Yaskawa INFORM job: A_ROOF_UPPER_0614_2_PAINT_36.JBI

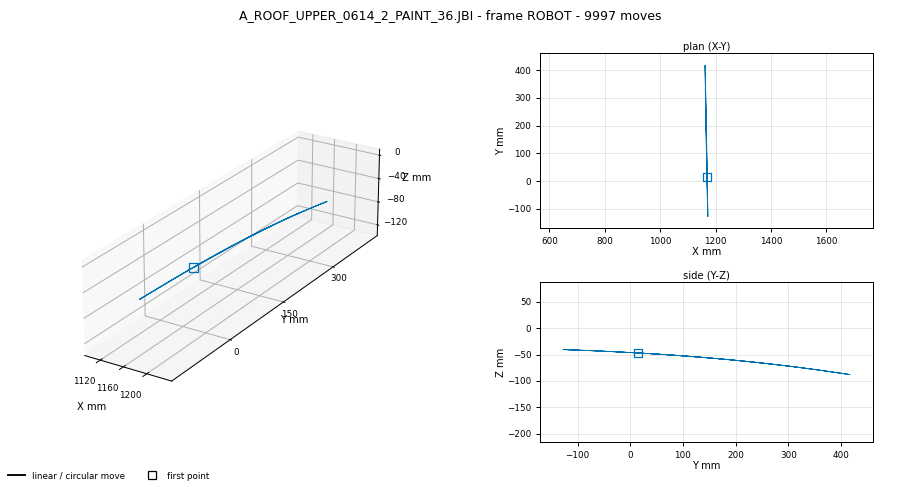
[picture p0: tool path of A_ROOF_UPPER_0614_2_PAINT_36.JBI in frame ROBOT, 9997 of 9997 moves have a stored position in this frame; points joined in program order, loops and branches not executed]
/JOB
//NAME A_ROOF_UPPER_0614_2_PAINT36
//POS
///NPOS 9997,0,0,0,0,0
///TOOL 1
///USER 0
///POSTYPE ROBOT
///RECTAN
///RCONF 1,0,0,0,0,0,0,0,0,0,0,0,0,0,0,0,0,0,0,0,0,0,0,0
C00000=1170.431,14.417,-46.796,-179.925,5.967,149.046
C00001=1170.426,14.666,-46.810,-179.923,5.968,149.045
C00002=1170.421,14.916,-46.824,-179.920,5.969,149.044
C00003=1170.416,15.166,-46.839,-179.918,5.970,149.044
C00004=1170.411,15.415,-46.853,-179.916,5.970,149.043
C00005=1170.405,15.664,-46.867,-179.913,5.970,149.043
C00006=1170.400,15.914,-46.881,-179.911,5.971,149.042
C00007=1170.396,16.164,-46.895,-179.908,5.973,149.042
C00008=1170.391,16.413,-46.910,-179.905,5.973,149.041
C00009=1170.386,16.663,-46.924,-179.903,5.974,149.040
C00010=1170.380,16.912,-46.938,-179.900,5.974,149.040
C00011=1170.375,17.161,-46.953,-179.898,5.975,149.039
C00012=1170.370,17.411,-46.967,-179.895,5.976,149.039
C00013=1170.366,17.661,-46.981,-179.893,5.977,149.038
C00014=1170.361,17.910,-46.996,-179.890,5.977,149.037
C00015=1170.356,18.160,-47.010,-179.887,5.978,149.037
C00016=1170.350,18.409,-47.024,-179.885,5.979,149.036
C00017=1170.345,18.659,-47.038,-179.882,5.980,149.036
C00018=1170.340,18.909,-47.052,-179.880,5.980,149.035
C00019=1170.334,19.159,-47.067,-179.878,5.981,149.034
C00020=1170.330,19.408,-47.082,-179.875,5.981,149.034
C00021=1170.325,19.657,-47.096,-179.873,5.982,149.033
C00022=1170.319,19.906,-47.110,-179.870,5.984,149.033
C00023=1170.314,20.156,-47.125,-179.867,5.984,149.032
C00024=1170.309,20.406,-47.139,-179.865,5.985,149.031
C00025=1170.304,20.656,-47.153,-179.862,5.985,149.031
C00026=1170.300,20.905,-47.168,-179.860,5.986,149.030
C00027=1170.295,21.154,-47.182,-179.857,5.987,149.030
C00028=1170.290,21.404,-47.197,-179.855,5.988,149.029
C00029=1170.284,21.653,-47.211,-179.852,5.989,149.029
C00030=1170.279,21.903,-47.226,-179.849,5.989,149.028
C00031=1170.274,22.152,-47.241,-179.847,5.990,149.027
C00032=1170.269,22.402,-47.255,-179.844,5.991,149.027
C00033=1170.264,22.652,-47.269,-179.842,5.991,149.026
C00034=1170.259,22.901,-47.283,-179.840,5.992,149.026
C00035=1170.254,23.151,-47.299,-179.836,5.993,149.025
C00036=1170.249,23.400,-47.313,-179.834,5.994,149.024
C00037=1170.244,23.650,-47.328,-179.832,5.995,149.024
C00038=1170.239,23.898,-47.342,-179.829,5.995,149.023
C00039=1170.234,24.148,-47.356,-179.827,5.996,149.023
C00040=1170.229,24.398,-47.371,-179.825,5.997,149.022
C00041=1170.223,24.647,-47.386,-179.821,5.998,149.022
C00042=1170.218,24.897,-47.401,-179.819,5.998,149.021
C00043=1170.213,25.147,-47.415,-179.817,5.999,149.020
C00044=1170.209,25.396,-47.430,-179.814,6.000,149.020
C00045=1170.203,25.646,-47.445,-179.812,6.001,149.019
C00046=1170.198,25.896,-47.459,-179.808,6.002,149.019
C00047=1170.193,26.145,-47.474,-179.806,6.002,149.018
C00048=1170.188,26.394,-47.488,-179.804,6.003,149.017
C00049=1170.183,26.644,-47.503,-179.801,6.004,149.017
C00050=1170.178,26.893,-47.518,-179.799,6.005,149.016
C00051=1170.173,27.143,-47.532,-179.796,6.006,149.016
C00052=1170.169,27.392,-47.547,-179.793,6.006,149.015
C00053=1170.163,27.642,-47.562,-179.791,6.007,149.015
C00054=1170.158,27.911,-47.578,-179.788,6.008,149.014
C00055=1170.153,28.180,-47.594,-179.785,6.009,149.013
C00056=1170.147,28.449,-47.610,-179.783,6.010,149.013
C00057=1170.141,28.717,-47.625,-179.780,6.010,149.012
C00058=1170.136,28.966,-47.640,-179.777,6.012,149.011
C00059=1170.131,29.216,-47.655,-179.775,6.012,149.011
C00060=1170.126,29.465,-47.670,-179.772,6.013,149.010
C00061=1170.121,29.715,-47.684,-179.769,6.013,149.010
C00062=1170.116,29.964,-47.700,-179.767,6.014,149.009
C00063=1170.111,30.215,-47.715,-179.764,6.016,149.008
C00064=1170.107,30.464,-47.730,-179.762,6.016,149.008
C00065=1170.101,30.714,-47.745,-179.759,6.017,149.007
C00066=1170.096,30.963,-47.760,-179.757,6.018,149.007
C00067=1170.091,31.213,-47.774,-179.754,6.018,149.006
C00068=1170.086,31.462,-47.789,-179.751,6.020,149.005
C00069=1170.081,31.712,-47.804,-179.749,6.020,149.005
C00070=1170.076,31.961,-47.819,-179.746,6.021,149.004
C00071=1170.071,32.210,-47.834,-179.744,6.022,149.004
C00072=1170.066,32.460,-47.849,-179.741,6.023,149.003
C00073=1170.061,32.709,-47.864,-179.739,6.024,149.003
C00074=1170.056,32.959,-47.878,-179.736,6.024,149.002
C00075=1170.050,33.209,-47.894,-179.734,6.025,149.001
C00076=1170.046,33.458,-47.909,-179.731,6.026,149.001
C00077=1170.040,33.708,-47.924,-179.728,6.027,149.000
C00078=1170.035,33.957,-47.939,-179.726,6.028,149.000
C00079=1170.031,34.206,-47.954,-179.723,6.028,148.999
C00080=1170.025,34.456,-47.969,-179.721,6.029,148.999
C00081=1170.021,34.706,-47.984,-179.718,6.030,148.998
C00082=1170.016,34.955,-48.000,-179.715,6.031,148.997
C00083=1170.011,35.205,-48.014,-179.713,6.032,148.997
C00084=1170.005,35.454,-48.030,-179.710,6.032,148.996
C00085=1170.001,35.703,-48.045,-179.708,6.034,148.996
C00086=1169.995,35.953,-48.060,-179.705,6.034,148.995
C00087=1169.990,36.202,-48.074,-179.703,6.035,148.995
C00088=1169.985,36.452,-48.090,-179.700,6.036,148.994
C00089=1169.980,36.701,-48.105,-179.698,6.037,148.994
C00090=1169.975,36.951,-48.121,-179.695,6.038,148.993
C00091=1169.970,37.201,-48.135,-179.692,6.038,148.992
C00092=1169.965,37.450,-48.151,-179.690,6.039,148.992
C00093=1169.960,37.699,-48.166,-179.687,6.041,148.991
C00094=1169.955,37.949,-48.181,-179.685,6.041,148.991
C00095=1169.950,38.198,-48.196,-179.682,6.042,148.990
C00096=1169.945,38.448,-48.211,-179.680,6.043,148.990
C00097=1169.940,38.698,-48.227,-179.677,6.044,148.989
C00098=1169.935,38.947,-48.242,-179.674,6.045,148.988
C00099=1169.930,39.196,-48.258,-179.672,6.045,148.988
C00100=1169.925,39.445,-48.273,-179.669,6.046,148.987
C00101=1169.920,39.695,-48.288,-179.666,6.048,148.987
C00102=1169.915,39.944,-48.303,-179.664,6.048,148.986
C00103=1169.910,40.195,-48.319,-179.662,6.049,148.985
C00104=1169.905,40.444,-48.334,-179.659,6.049,148.985
C00105=1169.900,40.693,-48.349,-179.656,6.051,148.984
C00106=1169.895,40.942,-48.365,-179.654,6.052,148.984
C00107=1169.889,41.192,-48.380,-179.652,6.052,148.983
C00108=1169.885,41.441,-48.395,-179.648,6.054,148.983
C00109=1169.880,41.691,-48.411,-179.646,6.054,148.982
C00110=1169.875,41.940,-48.426,-179.643,6.055,148.981
C00111=1169.870,42.190,-48.442,-179.641,6.056,148.981
C00112=1169.864,42.439,-48.457,-179.638,6.057,148.980
C00113=1169.860,42.689,-48.473,-179.635,6.058,148.980
C00114=1169.855,42.938,-48.488,-179.633,6.059,148.979
C00115=1169.849,43.188,-48.503,-179.630,6.060,148.979
C00116=1169.845,43.437,-48.518,-179.628,6.061,148.978
C00117=1169.840,43.686,-48.535,-179.625,6.061,148.977
C00118=1169.835,43.936,-48.551,-179.623,6.062,148.977
C00119=1169.830,44.185,-48.565,-179.620,6.063,148.976
C00120=1169.825,44.435,-48.581,-179.617,6.064,148.976
C00121=1169.819,44.684,-48.597,-179.615,6.065,148.975
C00122=1169.815,44.934,-48.613,-179.612,6.066,148.975
C00123=1169.810,45.183,-48.628,-179.610,6.067,148.974
C00124=1169.804,45.433,-48.643,-179.607,6.067,148.973
C00125=1169.800,45.683,-48.659,-179.605,6.068,148.973
C00126=1169.794,45.932,-48.675,-179.602,6.070,148.972
C00127=1169.790,46.181,-48.690,-179.600,6.071,148.972
C00128=1169.784,46.431,-48.705,-179.597,6.071,148.971
C00129=1169.779,46.681,-48.721,-179.594,6.073,148.971
C00130=1169.774,46.930,-48.737,-179.591,6.073,148.970
C00131=1169.770,47.179,-48.753,-179.589,6.074,148.970
C00132=1169.765,47.429,-48.769,-179.586,6.075,148.969
C00133=1169.760,47.678,-48.784,-179.583,6.076,148.968
C00134=1169.754,47.928,-48.800,-179.581,6.077,148.968
C00135=1169.750,48.177,-48.815,-179.578,6.078,148.967
C00136=1169.745,48.427,-48.831,-179.576,6.079,148.967
C00137=1169.740,48.676,-48.847,-179.573,6.079,148.966
C00138=1169.735,48.926,-48.863,-179.571,6.081,148.966
C00139=1169.730,49.175,-48.878,-179.568,6.082,148.965
C00140=1169.725,49.424,-48.893,-179.566,6.082,148.965
C00141=1169.720,49.674,-48.909,-179.563,6.084,148.964
C00142=1169.715,49.923,-48.926,-179.560,6.085,148.963
C00143=1169.710,50.172,-48.941,-179.558,6.085,148.963
C00144=1169.705,50.423,-48.957,-179.555,6.087,148.962
C00145=1169.699,50.672,-48.973,-179.552,6.087,148.962
C00146=1169.694,50.921,-48.989,-179.550,6.088,148.961
C00147=1169.690,51.171,-49.005,-179.547,6.089,148.961
C00148=1169.685,51.420,-49.020,-179.545,6.090,148.960
C00149=1169.680,51.669,-49.037,-179.542,6.091,148.959
C00150=1169.675,51.919,-49.052,-179.539,6.092,148.959
C00151=1169.670,52.168,-49.068,-179.537,6.093,148.958
C00152=1169.665,52.418,-49.085,-179.534,6.093,148.958
C00153=1169.660,52.667,-49.100,-179.531,6.095,148.957
C00154=1169.654,52.916,-49.116,-179.529,6.096,148.957
C00155=1169.650,53.166,-49.132,-179.527,6.097,148.956
C00156=1169.645,53.415,-49.148,-179.523,6.098,148.955
C00157=1169.640,53.665,-49.164,-179.521,6.099,148.955
C00158=1169.634,53.934,-49.181,-179.518,6.100,148.954
C00159=1169.629,54.202,-49.199,-179.515,6.101,148.954
C00160=1169.623,54.470,-49.216,-179.513,6.102,148.953
C00161=1169.618,54.739,-49.233,-179.510,6.103,148.953
C00162=1169.613,54.989,-49.249,-179.507,6.104,148.952
C00163=1169.609,55.238,-49.265,-179.505,6.105,148.951
C00164=1169.603,55.488,-49.281,-179.502,6.106,148.951
C00165=1169.598,55.737,-49.297,-179.499,6.107,148.950
C00166=1169.593,55.987,-49.313,-179.497,6.108,148.950
C00167=1169.588,56.235,-49.330,-179.494,6.108,148.949
C00168=1169.583,56.486,-49.346,-179.492,6.110,148.949
C00169=1169.578,56.734,-49.362,-179.489,6.111,148.948
C00170=1169.574,56.984,-49.378,-179.487,6.112,148.948
C00171=1169.568,57.233,-49.394,-179.484,6.113,148.947
C00172=1169.564,57.483,-49.410,-179.482,6.114,148.947
C00173=1169.559,57.732,-49.426,-179.478,6.115,148.946
C00174=1169.554,57.982,-49.442,-179.476,6.116,148.946
C00175=1169.549,58.231,-49.459,-179.474,6.116,148.945
C00176=1169.544,58.481,-49.475,-179.471,6.118,148.944
C00177=1169.539,58.730,-49.491,-179.468,6.119,148.944
C00178=1169.534,58.980,-49.507,-179.465,6.120,148.943
C00179=1169.529,59.229,-49.523,-179.463,6.121,148.943
C00180=1169.525,59.478,-49.540,-179.461,6.122,148.942
C00181=1169.519,59.728,-49.555,-179.457,6.123,148.942
C00182=1169.515,59.977,-49.572,-179.455,6.124,148.941
C00183=1169.509,60.227,-49.588,-179.453,6.124,148.940
C00184=1169.504,60.476,-49.605,-179.450,6.126,148.940
C00185=1169.499,60.725,-49.621,-179.447,6.127,148.939
C00186=1169.494,60.975,-49.637,-179.445,6.128,148.939
C00187=1169.489,61.224,-49.653,-179.442,6.129,148.938
C00188=1169.485,61.473,-49.670,-179.440,6.130,148.938
C00189=1169.479,61.723,-49.686,-179.437,6.131,148.937
C00190=1169.474,61.973,-49.703,-179.434,6.132,148.937
C00191=1169.469,62.221,-49.719,-179.431,6.133,148.936
C00192=1169.464,62.472,-49.735,-179.429,6.134,148.936
C00193=1169.460,62.721,-49.752,-179.426,6.135,148.935
C00194=1169.455,62.970,-49.768,-179.424,6.136,148.935
C00195=1169.450,63.219,-49.785,-179.421,6.137,148.934
C00196=1169.444,63.469,-49.801,-179.418,6.138,148.933
C00197=1169.440,63.719,-49.818,-179.416,6.139,148.933
C00198=1169.434,63.967,-49.834,-179.413,6.141,148.932
C00199=1169.430,64.217,-49.851,-179.410,6.141,148.932
C00200=1169.425,64.467,-49.867,-179.408,6.142,148.931
C00201=1169.419,64.716,-49.884,-179.405,6.143,148.931
C00202=1169.415,64.965,-49.900,-179.403,6.144,148.930
C00203=1169.410,65.215,-49.917,-179.400,6.145,148.929
C00204=1169.405,65.464,-49.933,-179.397,6.146,148.929
C00205=1169.400,65.714,-49.950,-179.394,6.148,148.928
C00206=1169.395,65.963,-49.966,-179.392,6.149,148.928
C00207=1169.390,66.212,-49.983,-179.390,6.149,148.927
C00208=1169.386,66.462,-49.999,-179.387,6.151,148.927
C00209=1169.380,66.711,-50.016,-179.385,6.152,148.926
C00210=1169.375,66.960,-50.033,-179.381,6.153,148.926
C00211=1169.371,67.210,-50.050,-179.379,6.154,148.925
C00212=1169.365,67.460,-50.066,-179.376,6.155,148.925
C00213=1169.360,67.709,-50.082,-179.374,6.156,148.924
C00214=1169.356,67.959,-50.099,-179.371,6.157,148.924
C00215=1169.351,68.207,-50.115,-179.368,6.158,148.923
C00216=1169.346,68.457,-50.133,-179.366,6.159,148.922
C00217=1169.341,68.707,-50.149,-179.363,6.160,148.922
C00218=1169.336,68.955,-50.166,-179.360,6.161,148.921
C00219=1169.331,69.205,-50.183,-179.358,6.163,148.921
C00220=1169.326,69.455,-50.200,-179.355,6.163,148.920
C00221=1169.321,69.704,-50.217,-179.352,6.165,148.920
C00222=1169.316,69.953,-50.233,-179.350,6.166,148.919
C00223=1169.312,70.203,-50.250,-179.347,6.167,148.919
C00224=1169.306,70.452,-50.267,-179.345,6.168,148.918
C00225=1169.301,70.701,-50.283,-179.342,6.168,148.918
C00226=1169.297,70.951,-50.300,-179.339,6.170,148.917
C00227=1169.291,71.200,-50.317,-179.337,6.171,148.917
C00228=1169.286,71.449,-50.334,-179.334,6.172,148.916
C00229=1169.281,71.699,-50.351,-179.331,6.173,148.915
C00230=1169.277,71.949,-50.368,-179.329,6.175,148.915
C00231=1169.271,72.198,-50.384,-179.326,6.175,148.914
C00232=1169.266,72.447,-50.401,-179.323,6.177,148.914
C00233=1169.262,72.697,-50.418,-179.321,6.178,148.914
C00234=1169.257,72.946,-50.436,-179.318,6.179,148.913
C00235=1169.252,73.195,-50.452,-179.316,6.180,148.912
C00236=1169.247,73.445,-50.469,-179.313,6.181,148.912
C00237=1169.242,73.694,-50.486,-179.310,6.182,148.911
C00238=1169.237,73.944,-50.503,-179.307,6.183,148.911
C00239=1169.232,74.193,-50.520,-179.305,6.184,148.910
C00240=1169.227,74.442,-50.537,-179.302,6.186,148.910
C00241=1169.223,74.691,-50.554,-179.300,6.186,148.909
C00242=1169.217,74.941,-50.572,-179.297,6.188,148.909
C00243=1169.212,75.190,-50.588,-179.294,6.189,148.908
C00244=1169.207,75.440,-50.605,-179.292,6.190,148.908
C00245=1169.203,75.689,-50.622,-179.289,6.191,148.907
C00246=1169.198,75.938,-50.640,-179.286,6.193,148.907
C00247=1169.193,76.188,-50.656,-179.284,6.193,148.906
C00248=1169.187,76.437,-50.673,-179.281,6.195,148.906
C00249=1169.183,76.686,-50.690,-179.279,6.196,148.905
C00250=1169.178,76.936,-50.708,-179.276,6.197,148.904
C00251=1169.174,77.185,-50.725,-179.273,6.198,148.904
C00252=1169.168,77.435,-50.742,-179.270,6.199,148.903
C00253=1169.163,77.685,-50.759,-179.268,6.200,148.903
C00254=1169.158,77.933,-50.776,-179.265,6.201,148.902
C00255=1169.153,78.183,-50.793,-179.263,6.202,148.902
C00256=1169.149,78.432,-50.810,-179.260,6.204,148.901
C00257=1169.144,78.681,-50.828,-179.257,6.205,148.901
C00258=1169.139,78.931,-50.845,-179.255,6.206,148.900
C00259=1169.134,79.181,-50.862,-179.252,6.207,148.900
C00260=1169.129,79.429,-50.880,-179.249,6.208,148.899
C00261=1169.124,79.678,-50.896,-179.247,6.209,148.899
C00262=1169.119,79.947,-50.915,-179.244,6.211,148.898
C00263=1169.114,80.216,-50.934,-179.241,6.212,148.898
C00264=1169.108,80.484,-50.953,-179.239,6.213,148.897
C00265=1169.103,80.752,-50.971,-179.235,6.214,148.896
C00266=1169.098,81.002,-50.989,-179.233,6.216,148.896
C00267=1169.093,81.251,-51.006,-179.230,6.216,148.895
C00268=1169.088,81.501,-51.023,-179.227,6.218,148.895
C00269=1169.083,81.750,-51.041,-179.225,6.219,148.894
C00270=1169.078,82.000,-51.058,-179.222,6.220,148.894
C00271=1169.073,82.248,-51.075,-179.220,6.221,148.893
C00272=1169.068,82.498,-51.092,-179.217,6.223,148.893
C00273=1169.063,82.747,-51.110,-179.214,6.223,148.892
C00274=1169.058,82.997,-51.128,-179.211,6.225,148.892
C00275=1169.054,83.246,-51.145,-179.209,6.226,148.891
C00276=1169.049,83.495,-51.162,-179.206,6.227,148.891
C00277=1169.044,83.745,-51.180,-179.203,6.229,148.890
C00278=1169.039,83.994,-51.197,-179.201,6.230,148.890
C00279=1169.034,84.243,-51.215,-179.198,6.231,148.889
C00280=1169.029,84.493,-51.232,-179.196,6.232,148.889
C00281=1169.024,84.742,-51.250,-179.193,6.234,148.888
C00282=1169.019,84.991,-51.268,-179.190,6.234,148.888
C00283=1169.015,85.241,-51.285,-179.188,6.236,148.887
C00284=1169.010,85.490,-51.303,-179.185,6.237,148.887
C00285=1169.005,85.740,-51.320,-179.182,6.238,148.886
C00286=1169.000,85.989,-51.338,-179.179,6.240,148.886
C00287=1168.995,86.238,-51.356,-179.177,6.240,148.885
C00288=1168.990,86.488,-51.373,-179.174,6.242,148.885
C00289=1168.985,86.737,-51.391,-179.172,6.243,148.884
C00290=1168.981,86.986,-51.409,-179.169,6.244,148.884
C00291=1168.975,87.236,-51.426,-179.167,6.245,148.883
C00292=1168.970,87.485,-51.444,-179.163,6.246,148.883
C00293=1168.966,87.734,-51.462,-179.161,6.248,148.882
C00294=1168.961,87.984,-51.478,-179.159,6.249,148.882
C00295=1168.956,88.233,-51.496,-179.155,6.250,148.881
C00296=1168.951,88.482,-51.514,-179.153,6.251,148.881
C00297=1168.946,88.732,-51.532,-179.151,6.253,148.880
C00298=1168.941,88.981,-51.550,-179.148,6.253,148.880
C00299=1168.936,89.230,-51.568,-179.145,6.255,148.879
C00300=1168.931,89.479,-51.586,-179.142,6.256,148.878
C00301=1168.926,89.729,-51.603,-179.140,6.257,148.878
C00302=1168.922,89.978,-51.620,-179.137,6.259,148.878
C00303=1168.917,90.227,-51.638,-179.134,6.260,148.877
C00304=1168.912,90.476,-51.656,-179.132,6.261,148.877
C00305=1168.907,90.725,-51.674,-179.129,6.263,148.876
C00306=1168.902,90.975,-51.691,-179.126,6.264,148.876
C00307=1168.897,91.224,-51.709,-179.124,6.265,148.875
C00308=1168.892,91.474,-51.727,-179.121,6.266,148.874
C00309=1168.887,91.723,-51.745,-179.118,6.267,148.874
C00310=1168.882,91.972,-51.763,-179.116,6.269,148.874
C00311=1168.877,92.221,-51.781,-179.113,6.270,148.873
C00312=1168.872,92.471,-51.799,-179.110,6.271,148.873
C00313=1168.868,92.721,-51.817,-179.108,6.272,148.872
C00314=1168.863,92.970,-51.835,-179.105,6.274,148.871
C00315=1168.858,93.219,-51.853,-179.102,6.275,148.871
C00316=1168.853,93.468,-51.871,-179.100,6.276,148.871
C00317=1168.848,93.718,-51.889,-179.097,6.278,148.870
C00318=1168.843,93.967,-51.907,-179.095,6.278,148.870
C00319=1168.838,94.216,-51.925,-179.092,6.280,148.869
C00320=1168.833,94.465,-51.943,-179.089,6.282,148.869
C00321=1168.829,94.714,-51.961,-179.087,6.282,148.868
C00322=1168.824,94.964,-51.979,-179.084,6.284,148.868
C00323=1168.819,95.213,-51.997,-179.081,6.285,148.867
C00324=1168.814,95.462,-52.015,-179.079,6.286,148.867
C00325=1168.810,95.712,-52.033,-179.075,6.288,148.866
C00326=1168.805,95.961,-52.051,-179.073,6.289,148.866
C00327=1168.800,96.210,-52.069,-179.071,6.290,148.865
C00328=1168.794,96.459,-52.088,-179.067,6.292,148.865
C00329=1168.790,96.709,-52.106,-179.065,6.293,148.864
C00330=1168.785,96.959,-52.124,-179.062,6.294,148.864
C00331=1168.780,97.208,-52.142,-179.059,6.296,148.863
C00332=1168.775,97.457,-52.160,-179.057,6.297,148.863
C00333=1168.770,97.706,-52.178,-179.054,6.298,148.862
C00334=1168.766,97.956,-52.196,-179.051,6.300,148.862
C00335=1168.761,98.205,-52.214,-179.049,6.300,148.861
C00336=1168.755,98.455,-52.233,-179.046,6.302,148.861
C00337=1168.751,98.703,-52.251,-179.044,6.303,148.860
C00338=1168.746,98.952,-52.269,-179.041,6.304,148.860
C00339=1168.741,99.202,-52.288,-179.038,6.306,148.859
C00340=1168.736,99.451,-52.306,-179.036,6.307,148.859
C00341=1168.732,99.701,-52.324,-179.033,6.308,148.858
C00342=1168.726,99.950,-52.342,-179.030,6.310,148.858
C00343=1168.721,100.199,-52.361,-179.028,6.311,148.857
C00344=1168.717,100.448,-52.379,-179.025,6.312,148.857
C00345=1168.712,100.698,-52.397,-179.022,6.314,148.856
C00346=1168.707,100.947,-52.415,-179.020,6.315,148.856
C00347=1168.702,101.196,-52.434,-179.017,6.316,148.855
C00348=1168.697,101.446,-52.453,-179.014,6.318,148.855
C00349=1168.693,101.695,-52.471,-179.012,6.319,148.854
C00350=1168.688,101.944,-52.489,-179.009,6.320,148.854
C00351=1168.682,102.193,-52.508,-179.006,6.322,148.853
C00352=1168.678,102.443,-52.527,-179.004,6.323,148.853
C00353=1168.673,102.692,-52.545,-179.001,6.324,148.852
C00354=1168.668,102.941,-52.563,-178.998,6.326,148.852
C00355=1168.663,103.191,-52.582,-178.996,6.327,148.851
C00356=1168.659,103.440,-52.600,-178.993,6.328,148.851
C00357=1168.654,103.689,-52.618,-178.990,6.330,148.850
C00358=1168.649,103.937,-52.637,-178.988,6.331,148.850
C00359=1168.644,104.188,-52.656,-178.985,6.333,148.850
C00360=1168.639,104.437,-52.674,-178.982,6.334,148.849
C00361=1168.634,104.685,-52.692,-178.979,6.336,148.849
C00362=1168.629,104.936,-52.711,-178.977,6.337,148.848
C00363=1168.624,105.185,-52.729,-178.974,6.338,148.848
C00364=1168.620,105.433,-52.748,-178.971,6.340,148.847
C00365=1168.615,105.684,-52.767,-178.969,6.340,148.847
C00366=1168.610,105.951,-52.787,-178.966,6.342,148.846
C00367=1168.604,106.220,-52.807,-178.963,6.344,148.846
C00368=1168.599,106.488,-52.827,-178.960,6.345,148.845
C00369=1168.594,106.757,-52.848,-178.957,6.347,148.845
C00370=1168.589,107.006,-52.866,-178.954,6.348,148.844
C00371=1168.584,107.255,-52.885,-178.952,6.349,148.844
C00372=1168.580,107.505,-52.903,-178.949,6.351,148.843
C00373=1168.575,107.754,-52.921,-178.946,6.352,148.843
C00374=1168.570,108.003,-52.941,-178.944,6.353,148.842
C00375=1168.565,108.252,-52.960,-178.941,6.355,148.842
C00376=1168.560,108.501,-52.978,-178.938,6.356,148.841
C00377=1168.556,108.751,-52.997,-178.936,6.358,148.841
C00378=1168.550,109.000,-53.016,-178.933,6.359,148.840
C00379=1168.546,109.249,-53.034,-178.930,6.360,148.840
C00380=1168.540,109.499,-53.053,-178.928,6.362,148.839
C00381=1168.536,109.747,-53.072,-178.925,6.364,148.839
C00382=1168.532,109.997,-53.090,-178.922,6.364,148.838
C00383=1168.526,110.246,-53.110,-178.920,6.366,148.838
C00384=1168.522,110.495,-53.128,-178.917,6.368,148.838
C00385=1168.517,110.745,-53.147,-178.915,6.369,148.837
C00386=1168.512,110.993,-53.166,-178.911,6.370,148.837
C00387=1168.507,111.243,-53.186,-178.909,6.372,148.836
C00388=1168.502,111.492,-53.204,-178.906,6.373,148.836
C00389=1168.498,111.742,-53.223,-178.903,6.374,148.835
C00390=1168.493,111.990,-53.242,-178.901,6.376,148.835
C00391=1168.488,112.240,-53.261,-178.898,6.377,148.834
C00392=1168.483,112.489,-53.280,-178.895,6.379,148.834
C00393=1168.478,112.738,-53.299,-178.893,6.380,148.833
C00394=1168.473,112.988,-53.318,-178.890,6.381,148.833
C00395=1168.468,113.237,-53.337,-178.887,6.383,148.832
C00396=1168.464,113.486,-53.356,-178.885,6.385,148.832
C00397=1168.459,113.735,-53.374,-178.882,6.385,148.831
C00398=1168.454,113.985,-53.394,-178.879,6.387,148.831
C00399=1168.449,114.234,-53.413,-178.876,6.389,148.831
C00400=1168.445,114.483,-53.432,-178.874,6.391,148.830
C00401=1168.439,114.732,-53.452,-178.872,6.391,148.830
C00402=1168.435,114.982,-53.470,-178.868,6.393,148.829
C00403=1168.430,115.231,-53.489,-178.866,6.395,148.829
C00404=1168.425,115.480,-53.509,-178.863,6.396,148.828
C00405=1168.420,115.729,-53.528,-178.861,6.397,148.828
C00406=1168.415,115.978,-53.547,-178.858,6.399,148.827
C00407=1168.410,116.228,-53.566,-178.855,6.400,148.827
C00408=1168.406,116.477,-53.585,-178.852,6.402,148.826
C00409=1168.400,116.726,-53.604,-178.850,6.403,148.826
C00410=1168.396,116.976,-53.624,-178.847,6.404,148.825
C00411=1168.391,117.224,-53.642,-178.844,6.406,148.825
C00412=1168.386,117.474,-53.662,-178.842,6.408,148.825
C00413=1168.381,117.723,-53.681,-178.839,6.409,148.824
C00414=1168.377,117.972,-53.701,-178.836,6.410,148.824
C00415=1168.372,118.221,-53.720,-178.833,6.412,148.823
C00416=1168.367,118.470,-53.739,-178.831,6.413,148.823
C00417=1168.362,118.720,-53.759,-178.828,6.415,148.822
C00418=1168.358,118.968,-53.778,-178.825,6.417,148.822
C00419=1168.353,119.219,-53.797,-178.823,6.417,148.821
C00420=1168.347,119.467,-53.816,-178.820,6.419,148.821
C00421=1168.343,119.717,-53.835,-178.817,6.421,148.821
C00422=1168.338,119.966,-53.855,-178.815,6.423,148.820
C00423=1168.333,120.215,-53.874,-178.812,6.423,148.820
C00424=1168.329,120.464,-53.894,-178.809,6.425,148.819
C00425=1168.323,120.713,-53.914,-178.807,6.427,148.819
C00426=1168.319,120.962,-53.933,-178.804,6.428,148.818
C00427=1168.315,121.212,-53.952,-178.801,6.430,148.818
C00428=1168.309,121.461,-53.972,-178.798,6.432,148.818
C00429=1168.304,121.710,-53.991,-178.796,6.432,148.817
C00430=1168.300,121.960,-54.011,-178.793,6.434,148.817
C00431=1168.295,122.208,-54.030,-178.790,6.436,148.816
C00432=1168.290,122.458,-54.049,-178.788,6.437,148.816
C00433=1168.285,122.707,-54.069,-178.785,6.439,148.815
C00434=1168.280,122.956,-54.088,-178.782,6.440,148.815
C00435=1168.276,123.205,-54.109,-178.780,6.441,148.814
C00436=1168.271,123.454,-54.128,-178.777,6.443,148.814
C00437=1168.266,123.703,-54.147,-178.774,6.445,148.813
C00438=1168.262,123.953,-54.167,-178.772,6.447,148.813
C00439=1168.256,124.202,-54.186,-178.769,6.447,148.812
C00440=1168.252,124.451,-54.206,-178.766,6.449,148.812
C00441=1168.247,124.700,-54.226,-178.764,6.451,148.812
C00442=1168.242,124.949,-54.245,-178.761,6.452,148.811
C00443=1168.237,125.199,-54.265,-178.758,6.454,148.811
C00444=1168.232,125.448,-54.285,-178.755,6.456,148.810
C00445=1168.228,125.697,-54.305,-178.753,6.456,148.810
C00446=1168.223,125.946,-54.324,-178.750,6.458,148.809
C00447=1168.219,126.195,-54.343,-178.747,6.460,148.809
C00448=1168.214,126.445,-54.363,-178.745,6.462,148.809
C00449=1168.209,126.693,-54.383,-178.742,6.463,148.808
C00450=1168.204,126.943,-54.403,-178.739,6.465,148.808
C00451=1168.199,127.192,-54.422,-178.736,6.466,148.807
C00452=1168.195,127.441,-54.443,-178.734,6.467,148.807
C00453=1168.190,127.690,-54.462,-178.731,6.469,148.806
C00454=1168.185,127.940,-54.482,-178.729,6.471,148.806
C00455=1168.180,128.189,-54.502,-178.726,6.473,148.806
C00456=1168.176,128.438,-54.522,-178.723,6.474,148.805
C00457=1168.170,128.687,-54.541,-178.720,6.476,148.805
C00458=1168.166,128.936,-54.561,-178.718,6.477,148.804
C00459=1168.161,129.186,-54.581,-178.715,6.478,148.804
C00460=1168.157,129.435,-54.601,-178.712,6.480,148.803
C00461=1168.151,129.683,-54.621,-178.710,6.482,148.803
C00462=1168.147,129.933,-54.640,-178.707,6.483,148.802
C00463=1168.142,130.182,-54.661,-178.704,6.485,148.802
C00464=1168.137,130.432,-54.680,-178.701,6.487,148.802
C00465=1168.133,130.680,-54.701,-178.698,6.488,148.801
C00466=1168.127,130.930,-54.721,-178.696,6.489,148.801
C00467=1168.122,131.179,-54.741,-178.694,6.491,148.800
C00468=1168.118,131.428,-54.761,-178.691,6.493,148.800
C00469=1168.113,131.677,-54.781,-178.688,6.494,148.799
C00470=1168.108,131.946,-54.802,-178.685,6.496,148.799
C00471=1168.103,132.215,-54.824,-178.682,6.498,148.799
C00472=1168.098,132.483,-54.846,-178.680,6.499,148.798
C00473=1168.092,132.752,-54.867,-178.676,6.501,148.798
C00474=1168.088,133.001,-54.888,-178.674,6.502,148.797
C00475=1168.083,133.250,-54.907,-178.671,6.504,148.797
C00476=1168.078,133.498,-54.927,-178.668,6.506,148.796
C00477=1168.073,133.748,-54.947,-178.666,6.508,148.796
C00478=1168.069,133.997,-54.967,-178.663,6.509,148.796
C00479=1168.064,134.246,-54.988,-178.660,6.511,148.795
C00480=1168.059,134.496,-55.008,-178.657,6.512,148.795
C00481=1168.055,134.745,-55.028,-178.654,6.514,148.794
C00482=1168.050,134.993,-55.048,-178.652,6.516,148.794
C00483=1168.045,135.243,-55.068,-178.649,6.517,148.794
C00484=1168.040,135.492,-55.089,-178.647,6.519,148.793
C00485=1168.035,135.741,-55.109,-178.644,6.520,148.793
C00486=1168.031,135.990,-55.129,-178.641,6.522,148.792
C00487=1168.026,136.239,-55.149,-178.639,6.524,148.792
C00488=1168.021,136.489,-55.170,-178.635,6.525,148.791
C00489=1168.016,136.738,-55.190,-178.633,6.527,148.791
C00490=1168.012,136.987,-55.210,-178.630,6.529,148.791
C00491=1168.007,137.235,-55.230,-178.627,6.530,148.790
C00492=1168.002,137.485,-55.251,-178.625,6.532,148.790
C00493=1167.997,137.734,-55.271,-178.622,6.534,148.789
C00494=1167.992,137.983,-55.291,-178.620,6.535,148.789
C00495=1167.988,138.232,-55.312,-178.617,6.536,148.789
C00496=1167.983,138.481,-55.333,-178.614,6.538,148.788
C00497=1167.978,138.730,-55.353,-178.612,6.540,148.788
C00498=1167.974,138.980,-55.373,-178.609,6.541,148.787
C00499=1167.968,139.229,-55.394,-178.606,6.543,148.787
C00500=1167.964,139.478,-55.414,-178.603,6.545,148.786
C00501=1167.960,139.727,-55.434,-178.600,6.547,148.786
C00502=1167.954,139.976,-55.455,-178.598,6.548,148.786
C00503=1167.950,140.225,-55.476,-178.595,6.550,148.785
C00504=1167.945,140.474,-55.496,-178.592,6.552,148.785
C00505=1167.940,140.724,-55.516,-178.590,6.554,148.785
C00506=1167.936,140.973,-55.537,-178.587,6.555,148.784
C00507=1167.931,141.222,-55.557,-178.584,6.557,148.784
C00508=1167.926,141.471,-55.578,-178.581,6.559,148.783
C00509=1167.922,141.720,-55.598,-178.579,6.560,148.783
C00510=1167.916,141.969,-55.619,-178.576,6.561,148.782
C00511=1167.912,142.218,-55.640,-178.573,6.563,148.782
C00512=1167.907,142.467,-55.660,-178.571,6.565,148.782
C00513=1167.902,142.717,-55.681,-178.568,6.566,148.781
C00514=1167.898,142.966,-55.701,-178.565,6.568,148.781
C00515=1167.893,143.215,-55.722,-178.563,6.570,148.780
C00516=1167.888,143.464,-55.743,-178.560,6.571,148.780
C00517=1167.883,143.713,-55.764,-178.557,6.573,148.780
C00518=1167.879,143.962,-55.784,-178.555,6.575,148.779
C00519=1167.874,144.211,-55.805,-178.552,6.577,148.779
C00520=1167.869,144.460,-55.826,-178.549,6.578,148.778
C00521=1167.865,144.709,-55.846,-178.546,6.580,148.778
C00522=1167.859,144.958,-55.867,-178.544,6.582,148.778
C00523=1167.855,145.207,-55.888,-178.541,6.584,148.777
C00524=1167.850,145.456,-55.909,-178.538,6.585,148.777
C00525=1167.846,145.706,-55.930,-178.536,6.587,148.777
C00526=1167.841,145.955,-55.951,-178.533,6.589,148.776
C00527=1167.837,146.204,-55.971,-178.530,6.590,148.776
C00528=1167.831,146.453,-55.992,-178.527,6.592,148.775
C00529=1167.826,146.702,-56.013,-178.524,6.594,148.775
C00530=1167.822,146.951,-56.033,-178.522,6.595,148.774
C00531=1167.817,147.200,-56.055,-178.519,6.597,148.774
C00532=1167.813,147.449,-56.075,-178.516,6.599,148.774
C00533=1167.807,147.698,-56.096,-178.514,6.601,148.773
C00534=1167.803,147.947,-56.117,-178.511,6.602,148.773
C00535=1167.799,148.196,-56.139,-178.508,6.604,148.773
C00536=1167.794,148.446,-56.160,-178.506,6.606,148.772
C00537=1167.789,148.695,-56.180,-178.503,6.608,148.772
C00538=1167.784,148.944,-56.201,-178.500,6.609,148.771
C00539=1167.780,149.192,-56.222,-178.497,6.611,148.771
C00540=1167.775,149.441,-56.243,-178.495,6.613,148.771
C00541=1167.769,149.691,-56.264,-178.492,6.615,148.770
C00542=1167.766,149.940,-56.285,-178.489,6.616,148.770
C00543=1167.761,150.189,-56.306,-178.487,6.618,148.769
C00544=1167.756,150.438,-56.327,-178.484,6.620,148.769
C00545=1167.751,150.687,-56.348,-178.481,6.622,148.769
C00546=1167.746,150.936,-56.369,-178.479,6.623,148.768
C00547=1167.741,151.185,-56.390,-178.476,6.625,148.768
C00548=1167.737,151.435,-56.411,-178.473,6.627,148.768
C00549=1167.732,151.683,-56.433,-178.470,6.629,148.767
C00550=1167.727,151.933,-56.454,-178.468,6.630,148.767
C00551=1167.723,152.181,-56.475,-178.465,6.632,148.766
C00552=1167.718,152.430,-56.496,-178.462,6.634,148.766
C00553=1167.713,152.680,-56.517,-178.460,6.636,148.766
C00554=1167.708,152.929,-56.539,-178.457,6.637,148.765
C00555=1167.704,153.178,-56.559,-178.454,6.639,148.765
C00556=1167.699,153.426,-56.581,-178.452,6.641,148.765
C00557=1167.694,153.676,-56.602,-178.449,6.643,148.764
C00558=1167.690,153.925,-56.624,-178.446,6.644,148.764
C00559=1167.685,154.174,-56.644,-178.444,6.646,148.763
C00560=1167.680,154.423,-56.666,-178.441,6.648,148.763
C00561=1167.675,154.672,-56.687,-178.438,6.650,148.763
C00562=1167.671,154.921,-56.709,-178.435,6.651,148.762
C00563=1167.666,155.171,-56.730,-178.433,6.653,148.762
C00564=1167.662,155.419,-56.751,-178.430,6.655,148.762
C00565=1167.656,155.668,-56.772,-178.427,6.657,148.761
C00566=1167.652,155.917,-56.794,-178.425,6.658,148.761
C00567=1167.647,156.166,-56.816,-178.421,6.661,148.760
C00568=1167.642,156.415,-56.837,-178.419,6.663,148.760
C00569=1167.638,156.665,-56.859,-178.416,6.664,148.760
C00570=1167.633,156.914,-56.879,-178.413,6.666,148.759
C00571=1167.629,157.162,-56.901,-178.411,6.668,148.759
C00572=1167.624,157.411,-56.923,-178.408,6.670,148.759
C00573=1167.619,157.661,-56.944,-178.405,6.671,148.758
C00574=1167.615,157.929,-56.967,-178.403,6.673,148.758
C00575=1167.609,158.199,-56.991,-178.399,6.676,148.757
C00576=1167.604,158.468,-57.013,-178.397,6.677,148.757
C00577=1167.598,158.736,-57.036,-178.394,6.679,148.757
C00578=1167.594,158.986,-57.059,-178.391,6.681,148.756
C00579=1167.589,159.234,-57.080,-178.389,6.683,148.756
C00580=1167.584,159.483,-57.102,-178.386,6.684,148.756
C00581=1167.580,159.733,-57.123,-178.383,6.686,148.755
C00582=1167.575,159.982,-57.145,-178.380,6.689,148.755
C00583=1167.571,160.231,-57.167,-178.377,6.691,148.754
C00584=1167.566,160.480,-57.189,-178.374,6.692,148.754
C00585=1167.561,160.729,-57.209,-178.372,6.694,148.754
C00586=1167.557,160.978,-57.231,-178.369,6.696,148.753
C00587=1167.552,161.227,-57.253,-178.366,6.698,148.753
C00588=1167.547,161.475,-57.274,-178.364,6.699,148.753
C00589=1167.543,161.724,-57.296,-178.361,6.701,148.752
C00590=1167.538,161.973,-57.318,-178.358,6.703,148.752
C00591=1167.534,162.223,-57.339,-178.356,6.705,148.751
C00592=1167.529,162.472,-57.361,-178.353,6.707,148.751
C00593=1167.524,162.720,-57.383,-178.350,6.709,148.751
C00594=1167.520,162.970,-57.405,-178.347,6.711,148.751
C00595=1167.514,163.219,-57.427,-178.345,6.713,148.750
C00596=1167.510,163.468,-57.449,-178.342,6.714,148.750
C00597=1167.505,163.717,-57.471,-178.339,6.716,148.749
C00598=1167.501,163.966,-57.493,-178.337,6.718,148.749
C00599=1167.496,164.215,-57.515,-178.334,6.720,148.749
C00600=1167.491,164.463,-57.536,-178.331,6.721,148.748
C00601=1167.487,164.713,-57.558,-178.329,6.723,148.748
C00602=1167.482,164.961,-57.580,-178.326,6.725,148.748
C00603=1167.477,165.211,-57.602,-178.323,6.728,148.747
C00604=1167.473,165.459,-57.624,-178.320,6.729,148.747
C00605=1167.468,165.709,-57.646,-178.318,6.731,148.747
C00606=1167.463,165.957,-57.668,-178.315,6.733,148.746
C00607=1167.458,166.207,-57.690,-178.312,6.735,148.746
C00608=1167.454,166.455,-57.712,-178.310,6.737,148.746
C00609=1167.449,166.705,-57.734,-178.307,6.738,148.745
C00610=1167.444,166.953,-57.756,-178.304,6.740,148.745
C00611=1167.440,167.203,-57.778,-178.301,6.743,148.745
C00612=1167.435,167.451,-57.799,-178.298,6.744,148.744
C00613=1167.430,167.701,-57.822,-178.296,6.746,148.744
C00614=1167.425,167.950,-57.844,-178.293,6.748,148.744
C00615=1167.421,168.199,-57.866,-178.291,6.750,148.743
C00616=1167.417,168.447,-57.888,-178.288,6.752,148.743
C00617=1167.412,168.696,-57.910,-178.285,6.754,148.743
C00618=1167.407,168.945,-57.932,-178.282,6.756,148.742
C00619=1167.402,169.195,-57.954,-178.279,6.758,148.742
C00620=1167.398,169.443,-57.976,-178.277,6.760,148.741
C00621=1167.393,169.693,-57.998,-178.274,6.761,148.741
C00622=1167.388,169.941,-58.021,-178.271,6.763,148.741
C00623=1167.384,170.190,-58.043,-178.269,6.765,148.741
C00624=1167.379,170.439,-58.065,-178.266,6.767,148.740
C00625=1167.375,170.688,-58.087,-178.263,6.770,148.740
C00626=1167.369,170.937,-58.110,-178.261,6.771,148.739
C00627=1167.365,171.186,-58.132,-178.258,6.773,148.739
C00628=1167.361,171.435,-58.154,-178.255,6.775,148.739
C00629=1167.355,171.684,-58.176,-178.252,6.777,148.738
C00630=1167.351,171.933,-58.199,-178.250,6.779,148.738
C00631=1167.346,172.182,-58.221,-178.247,6.781,148.738
C00632=1167.341,172.431,-58.243,-178.244,6.783,148.738
C00633=1167.337,172.680,-58.266,-178.242,6.785,148.737
C00634=1167.332,172.929,-58.288,-178.239,6.787,148.737
C00635=1167.327,173.178,-58.311,-178.236,6.788,148.736
C00636=1167.323,173.426,-58.333,-178.234,6.790,148.736
C00637=1167.319,173.676,-58.355,-178.231,6.793,148.736
C00638=1167.314,173.925,-58.378,-178.228,6.795,148.736
C00639=1167.309,174.173,-58.400,-178.225,6.797,148.735
C00640=1167.305,174.423,-58.422,-178.223,6.798,148.735
C00641=1167.300,174.672,-58.445,-178.220,6.800,148.734
C00642=1167.295,174.920,-58.467,-178.217,6.803,148.734
C00643=1167.291,175.169,-58.490,-178.214,6.804,148.734
C00644=1167.286,175.418,-58.512,-178.212,6.807,148.734
C00645=1167.281,175.667,-58.535,-178.209,6.808,148.733
C00646=1167.277,175.916,-58.558,-178.206,6.810,148.733
C00647=1167.272,176.164,-58.580,-178.203,6.813,148.733
C00648=1167.267,176.414,-58.603,-178.201,6.814,148.732
C00649=1167.263,176.663,-58.625,-178.198,6.817,148.732
C00650=1167.258,176.913,-58.648,-178.196,6.818,148.732
C00651=1167.254,177.161,-58.670,-178.193,6.820,148.731
C00652=1167.249,177.410,-58.693,-178.190,6.823,148.731
C00653=1167.245,177.659,-58.716,-178.187,6.824,148.731
C00654=1167.239,177.908,-58.738,-178.184,6.826,148.730
C00655=1167.235,178.157,-58.761,-178.182,6.828,148.730
C00656=1167.230,178.406,-58.784,-178.179,6.830,148.730
C00657=1167.226,178.654,-58.806,-178.176,6.833,148.729
C00658=1167.221,178.903,-58.829,-178.174,6.834,148.729
C00659=1167.217,179.153,-58.851,-178.171,6.836,148.729
C00660=1167.212,179.402,-58.875,-178.169,6.838,148.729
C00661=1167.207,179.650,-58.897,-178.166,6.840,148.728
C00662=1167.202,179.899,-58.920,-178.163,6.843,148.728
C00663=1167.198,180.148,-58.943,-178.160,6.844,148.727
C00664=1167.194,180.397,-58.966,-178.157,6.846,148.727
C00665=1167.188,180.645,-58.989,-178.155,6.848,148.727
C00666=1167.184,180.895,-59.011,-178.152,6.851,148.727
C00667=1167.179,181.144,-59.034,-178.149,6.853,148.726
C00668=1167.175,181.393,-59.057,-178.146,6.854,148.726
C00669=1167.171,181.642,-59.080,-178.144,6.856,148.726
C00670=1167.165,181.890,-59.103,-178.141,6.859,148.725
C00671=1167.161,182.139,-59.125,-178.138,6.861,148.725
C00672=1167.156,182.388,-59.149,-178.136,6.863,148.725
C00673=1167.152,182.637,-59.172,-178.133,6.864,148.724
C00674=1167.147,182.886,-59.194,-178.130,6.867,148.724
C00675=1167.142,183.135,-59.217,-178.128,6.869,148.724
C00676=1167.137,183.384,-59.240,-178.125,6.871,148.724
C00677=1167.133,183.633,-59.263,-178.122,6.873,148.723
C00678=1167.128,183.902,-59.288,-178.119,6.875,148.723
C00679=1167.123,184.172,-59.313,-178.116,6.877,148.722
C00680=1167.118,184.442,-59.338,-178.113,6.879,148.722
C00681=1167.113,184.711,-59.364,-178.111,6.882,148.722
C00682=1167.108,184.960,-59.386,-178.107,6.884,148.722
C00683=1167.104,185.209,-59.409,-178.105,6.886,148.721
C00684=1167.100,185.458,-59.432,-178.102,6.888,148.721
C00685=1167.094,185.707,-59.455,-178.100,6.890,148.721
C00686=1167.090,185.956,-59.479,-178.097,6.892,148.720
C00687=1167.086,186.204,-59.501,-178.094,6.894,148.720
C00688=1167.081,186.453,-59.525,-178.091,6.896,148.720
C00689=1167.076,186.702,-59.548,-178.089,6.899,148.720
C00690=1167.072,186.951,-59.571,-178.086,6.901,148.719
C00691=1167.068,187.200,-59.594,-178.083,6.902,148.719
C00692=1167.063,187.449,-59.618,-178.080,6.904,148.719
C00693=1167.058,187.698,-59.641,-178.078,6.907,148.718
C00694=1167.053,187.947,-59.664,-178.075,6.909,148.718
C00695=1167.048,188.196,-59.687,-178.072,6.911,148.718
C00696=1167.044,188.444,-59.710,-178.070,6.912,148.717
C00697=1167.039,188.693,-59.733,-178.067,6.915,148.717
C00698=1167.035,188.942,-59.757,-178.064,6.917,148.717
C00699=1167.030,189.191,-59.781,-178.062,6.919,148.717
C00700=1167.026,189.440,-59.804,-178.058,6.921,148.716
C00701=1167.021,189.689,-59.828,-178.056,6.924,148.716
C00702=1167.016,189.938,-59.851,-178.053,6.925,148.716
C00703=1167.012,190.187,-59.874,-178.050,6.928,148.715
C00704=1167.008,190.436,-59.897,-178.048,6.930,148.715
C00705=1167.003,190.684,-59.921,-178.045,6.932,148.715
C00706=1166.999,190.933,-59.944,-178.043,6.934,148.715
C00707=1166.994,191.182,-59.968,-178.039,6.936,148.714
C00708=1166.989,191.431,-59.991,-178.037,6.938,148.714
C00709=1166.984,191.679,-60.014,-178.034,6.940,148.714
C00710=1166.979,191.928,-60.038,-178.031,6.943,148.713
C00711=1166.975,192.177,-60.062,-178.029,6.945,148.713
C00712=1166.970,192.426,-60.085,-178.026,6.946,148.713
C00713=1166.965,192.675,-60.108,-178.023,6.949,148.713
C00714=1166.961,192.923,-60.132,-178.021,6.951,148.713
C00715=1166.956,193.172,-60.156,-178.018,6.953,148.712
C00716=1166.952,193.421,-60.179,-178.015,6.956,148.712
C00717=1166.947,193.670,-60.203,-178.012,6.957,148.711
C00718=1166.942,193.919,-60.227,-178.010,6.959,148.711
C00719=1166.938,194.168,-60.250,-178.007,6.962,148.711
C00720=1166.934,194.417,-60.274,-178.004,6.964,148.711
C00721=1166.929,194.666,-60.298,-178.002,6.966,148.711
C00722=1166.925,194.915,-60.321,-177.999,6.968,148.710
C00723=1166.920,195.164,-60.345,-177.996,6.970,148.710
C00724=1166.915,195.413,-60.369,-177.994,6.972,148.710
C00725=1166.911,195.661,-60.393,-177.991,6.975,148.709
C00726=1166.906,195.910,-60.416,-177.988,6.977,148.709
C00727=1166.902,196.159,-60.439,-177.986,6.979,148.709
C00728=1166.897,196.407,-60.463,-177.982,6.981,148.709
C00729=1166.893,196.656,-60.487,-177.980,6.983,148.708
C00730=1166.887,196.905,-60.511,-177.978,6.985,148.708
C00731=1166.883,197.154,-60.535,-177.974,6.988,148.708
C00732=1166.878,197.403,-60.559,-177.972,6.990,148.707
C00733=1166.874,197.652,-60.582,-177.969,6.992,148.707
C00734=1166.869,197.900,-60.606,-177.966,6.994,148.707
C00735=1166.865,198.150,-60.630,-177.963,6.996,148.707
C00736=1166.861,198.398,-60.654,-177.961,6.998,148.706
C00737=1166.856,198.647,-60.678,-177.958,7.001,148.706
C00738=1166.851,198.896,-60.702,-177.955,7.003,148.706
C00739=1166.847,199.144,-60.726,-177.953,7.005,148.706
C00740=1166.842,199.393,-60.750,-177.950,7.007,148.705
C00741=1166.837,199.642,-60.774,-177.948,7.009,148.705
C00742=1166.833,199.890,-60.798,-177.944,7.012,148.705
C00743=1166.829,200.140,-60.821,-177.942,7.014,148.705
C00744=1166.824,200.389,-60.846,-177.940,7.016,148.704
C00745=1166.819,200.638,-60.869,-177.936,7.019,148.704
C00746=1166.815,200.886,-60.894,-177.934,7.020,148.704
C00747=1166.810,201.135,-60.918,-177.931,7.022,148.704
C00748=1166.805,201.383,-60.942,-177.928,7.025,148.703
C00749=1166.801,201.633,-60.966,-177.926,7.027,148.703
C00750=1166.797,201.881,-60.990,-177.923,7.030,148.703
C00751=1166.792,202.130,-61.014,-177.920,7.032,148.703
C00752=1166.787,202.379,-61.038,-177.918,7.034,148.702
C00753=1166.782,202.628,-61.062,-177.915,7.036,148.702
C00754=1166.779,202.877,-61.087,-177.912,7.038,148.702
C00755=1166.774,203.125,-61.111,-177.910,7.040,148.702
C00756=1166.769,203.374,-61.135,-177.906,7.043,148.701
C00757=1166.764,203.623,-61.159,-177.904,7.045,148.701
C00758=1166.760,203.871,-61.183,-177.901,7.047,148.701
C00759=1166.756,204.121,-61.208,-177.898,7.049,148.700
C00760=1166.751,204.369,-61.232,-177.896,7.051,148.700
C00761=1166.747,204.618,-61.256,-177.893,7.054,148.700
C00762=1166.741,204.867,-61.280,-177.891,7.056,148.700
C00763=1166.738,205.116,-61.304,-177.887,7.059,148.700
C00764=1166.733,205.364,-61.328,-177.885,7.060,148.699
C00765=1166.728,205.613,-61.353,-177.883,7.063,148.699
C00766=1166.724,205.862,-61.377,-177.879,7.065,148.699
C00767=1166.719,206.111,-61.402,-177.877,7.067,148.699
C00768=1166.715,206.359,-61.426,-177.874,7.070,148.698
C00769=1166.710,206.608,-61.451,-177.871,7.072,148.698
C00770=1166.705,206.857,-61.475,-177.868,7.075,148.698
C00771=1166.701,207.106,-61.499,-177.866,7.076,148.698
C00772=1166.696,207.354,-61.524,-177.864,7.078,148.697
C00773=1166.692,207.603,-61.548,-177.860,7.081,148.697
C00774=1166.687,207.852,-61.573,-177.858,7.083,148.697
C00775=1166.683,208.101,-61.597,-177.855,7.086,148.697
C00776=1166.678,208.349,-61.622,-177.852,7.088,148.696
C00777=1166.674,208.598,-61.646,-177.849,7.090,148.696
C00778=1166.669,208.847,-61.671,-177.847,7.092,148.696
C00779=1166.664,209.096,-61.695,-177.845,7.094,148.696
C00780=1166.660,209.345,-61.720,-177.841,7.097,148.695
C00781=1166.656,209.593,-61.744,-177.839,7.099,148.695
C00782=1166.650,209.864,-61.771,-177.836,7.102,148.695
C00783=1166.646,210.134,-61.798,-177.833,7.104,148.695
C00784=1166.641,210.405,-61.825,-177.830,7.107,148.695
C00785=1166.636,210.675,-61.852,-177.827,7.109,148.694
C00786=1166.631,210.924,-61.877,-177.824,7.112,148.694
C00787=1166.627,211.173,-61.901,-177.822,7.114,148.694
C00788=1166.621,211.421,-61.925,-177.819,7.116,148.694
C00789=1166.618,211.670,-61.950,-177.816,7.118,148.693
C00790=1166.613,211.919,-61.975,-177.813,7.121,148.693
C00791=1166.609,212.168,-62.000,-177.811,7.123,148.693
C00792=1166.604,212.416,-62.024,-177.808,7.125,148.693
C00793=1166.599,212.665,-62.049,-177.805,7.128,148.693
C00794=1166.595,212.914,-62.074,-177.803,7.130,148.692
C00795=1166.590,213.162,-62.099,-177.800,7.133,148.692
C00796=1166.586,213.412,-62.124,-177.797,7.134,148.692
C00797=1166.581,213.660,-62.148,-177.795,7.137,148.692
C00798=1166.576,213.908,-62.173,-177.792,7.139,148.691
C00799=1166.573,214.157,-62.198,-177.789,7.142,148.691
C00800=1166.568,214.406,-62.222,-177.786,7.144,148.691
C00801=1166.563,214.655,-62.248,-177.783,7.146,148.691
C00802=1166.559,214.903,-62.272,-177.781,7.149,148.691
C00803=1166.554,215.153,-62.297,-177.778,7.151,148.690
C00804=1166.550,215.401,-62.323,-177.776,7.153,148.690
C00805=1166.545,215.650,-62.348,-177.772,7.156,148.690
C00806=1166.541,215.898,-62.372,-177.770,7.158,148.690
C00807=1166.536,216.148,-62.397,-177.767,7.161,148.689
C00808=1166.531,216.396,-62.422,-177.765,7.163,148.689
C00809=1166.528,216.645,-62.447,-177.761,7.165,148.689
C00810=1166.523,216.893,-62.472,-177.759,7.167,148.689
C00811=1166.518,217.142,-62.498,-177.756,7.170,148.688
C00812=1166.513,217.391,-62.522,-177.754,7.172,148.688
C00813=1166.510,217.639,-62.547,-177.751,7.175,148.688
C00814=1166.505,217.888,-62.572,-177.748,7.177,148.688
C00815=1166.500,218.137,-62.598,-177.745,7.180,148.688
C00816=1166.495,218.386,-62.623,-177.743,7.182,148.688
C00817=1166.491,218.635,-62.648,-177.740,7.185,148.687
C00818=1166.487,218.883,-62.672,-177.738,7.186,148.687
C00819=1166.482,219.132,-62.698,-177.735,7.189,148.687
C00820=1166.477,219.380,-62.723,-177.732,7.191,148.687
C00821=1166.473,219.629,-62.749,-177.729,7.194,148.687
C00822=1166.468,219.877,-62.774,-177.727,7.196,148.686
C00823=1166.464,220.127,-62.799,-177.724,7.199,148.686
C00824=1166.460,220.375,-62.824,-177.721,7.201,148.686
C00825=1166.455,220.623,-62.850,-177.718,7.203,148.686
C00826=1166.451,220.873,-62.875,-177.716,7.205,148.685
C00827=1166.446,221.121,-62.900,-177.713,7.208,148.685
C00828=1166.442,221.370,-62.926,-177.710,7.210,148.685
C00829=1166.437,221.618,-62.950,-177.708,7.213,148.685
C00830=1166.432,221.867,-62.976,-177.705,7.215,148.685
C00831=1166.428,222.115,-63.002,-177.702,7.218,148.684
C00832=1166.423,222.365,-63.027,-177.700,7.220,148.684
C00833=1166.420,222.613,-63.052,-177.697,7.222,148.684
C00834=1166.415,222.861,-63.077,-177.695,7.225,148.684
C00835=1166.411,223.110,-63.103,-177.691,7.227,148.684
C00836=1166.405,223.359,-63.128,-177.689,7.230,148.684
C00837=1166.401,223.608,-63.153,-177.686,7.232,148.683
C00838=1166.397,223.857,-63.179,-177.683,7.235,148.683
C00839=1166.392,224.105,-63.204,-177.681,7.237,148.683
C00840=1166.388,224.353,-63.230,-177.678,7.240,148.683
C00841=1166.383,224.603,-63.255,-177.675,7.242,148.683
C00842=1166.379,224.851,-63.281,-177.672,7.244,148.682
C00843=1166.374,225.100,-63.306,-177.670,7.246,148.682
C00844=1166.370,225.349,-63.332,-177.667,7.249,148.682
C00845=1166.365,225.597,-63.357,-177.665,7.251,148.682
C00846=1166.361,225.845,-63.383,-177.662,7.254,148.682
C00847=1166.357,226.094,-63.409,-177.659,7.257,148.681
C00848=1166.352,226.342,-63.434,-177.656,7.259,148.681
C00849=1166.347,226.592,-63.460,-177.653,7.261,148.681
C00850=1166.343,226.841,-63.486,-177.651,7.264,148.681
C00851=1166.338,227.089,-63.511,-177.648,7.267,148.681
C00852=1166.334,227.338,-63.537,-177.646,7.268,148.680
C00853=1166.329,227.587,-63.563,-177.643,7.271,148.680
C00854=1166.324,227.835,-63.588,-177.640,7.274,148.680
C00855=1166.320,228.084,-63.614,-177.637,7.276,148.680
C00856=1166.316,228.332,-63.639,-177.635,7.279,148.680
C00857=1166.312,228.581,-63.665,-177.632,7.281,148.680
C00858=1166.306,228.830,-63.691,-177.629,7.284,148.679
C00859=1166.302,229.078,-63.718,-177.626,7.286,148.679
C00860=1166.298,229.327,-63.743,-177.624,7.288,148.679
C00861=1166.294,229.575,-63.769,-177.621,7.291,148.679
C00862=1166.289,229.823,-63.795,-177.618,7.293,148.679
C00863=1166.285,230.072,-63.820,-177.616,7.296,148.679
C00864=1166.280,230.321,-63.847,-177.613,7.299,148.678
C00865=1166.276,230.570,-63.872,-177.610,7.301,148.678
C00866=1166.271,230.818,-63.898,-177.607,7.304,148.678
C00867=1166.267,231.067,-63.924,-177.605,7.306,148.678
C00868=1166.263,231.315,-63.950,-177.602,7.309,148.678
C00869=1166.258,231.564,-63.976,-177.599,7.311,148.678
C00870=1166.253,231.813,-64.002,-177.597,7.313,148.677
C00871=1166.249,232.061,-64.028,-177.594,7.316,148.677
C00872=1166.244,232.310,-64.053,-177.592,7.318,148.677
C00873=1166.240,232.559,-64.080,-177.588,7.321,148.677
C00874=1166.236,232.807,-64.106,-177.586,7.324,148.677
C00875=1166.231,233.056,-64.132,-177.583,7.326,148.677
C00876=1166.226,233.304,-64.157,-177.580,7.329,148.676
C00877=1166.222,233.553,-64.184,-177.578,7.331,148.676
C00878=1166.218,233.802,-64.210,-177.575,7.334,148.676
C00879=1166.213,234.050,-64.236,-177.572,7.336,148.676
C00880=1166.209,234.299,-64.263,-177.570,7.338,148.676
C00881=1166.204,234.548,-64.289,-177.567,7.341,148.676
C00882=1166.200,234.796,-64.314,-177.564,7.344,148.675
C00883=1166.195,235.044,-64.341,-177.562,7.346,148.675
C00884=1166.191,235.293,-64.367,-177.559,7.349,148.675
C00885=1166.187,235.542,-64.393,-177.556,7.351,148.675
C00886=1166.181,235.814,-64.422,-177.553,7.354,148.675
C00887=1166.177,236.085,-64.451,-177.551,7.357,148.675
C00888=1166.172,236.357,-64.479,-177.547,7.359,148.674
C00889=1166.167,236.628,-64.508,-177.545,7.362,148.674
C00890=1166.163,236.877,-64.534,-177.541,7.365,148.674
C00891=1166.158,237.126,-64.561,-177.539,7.368,148.674
C00892=1166.154,237.374,-64.587,-177.536,7.370,148.674
C00893=1166.149,237.622,-64.613,-177.534,7.373,148.674
C00894=1166.145,237.871,-64.639,-177.530,7.376,148.673
C00895=1166.140,238.120,-64.666,-177.528,7.378,148.673
C00896=1166.136,238.368,-64.692,-177.526,7.381,148.673
C00897=1166.131,238.617,-64.719,-177.522,7.383,148.673
C00898=1166.127,238.866,-64.745,-177.520,7.385,148.673
C00899=1166.122,239.114,-64.772,-177.517,7.388,148.673
C00900=1166.118,239.363,-64.797,-177.515,7.391,148.673
C00901=1166.113,239.611,-64.825,-177.512,7.393,148.672
C00902=1166.109,239.860,-64.851,-177.509,7.396,148.672
C00903=1166.104,240.109,-64.877,-177.506,7.399,148.672
C00904=1166.101,240.357,-64.904,-177.504,7.401,148.672
C00905=1166.096,240.606,-64.930,-177.501,7.404,148.672
C00906=1166.092,240.854,-64.957,-177.498,7.407,148.672
C00907=1166.087,241.103,-64.984,-177.496,7.409,148.672
C00908=1166.083,241.352,-65.009,-177.493,7.412,148.672
C00909=1166.078,241.600,-65.037,-177.490,7.414,148.671
C00910=1166.074,241.848,-65.063,-177.488,7.417,148.671
C00911=1166.070,242.097,-65.090,-177.485,7.419,148.671
C00912=1166.065,242.346,-65.116,-177.482,7.422,148.671
C00913=1166.061,242.594,-65.143,-177.480,7.424,148.671
C00914=1166.056,242.842,-65.170,-177.477,7.427,148.671
C00915=1166.052,243.091,-65.196,-177.474,7.430,148.671
C00916=1166.047,243.340,-65.223,-177.472,7.432,148.671
C00917=1166.042,243.588,-65.250,-177.469,7.435,148.670
C00918=1166.039,243.836,-65.276,-177.466,7.438,148.670
C00919=1166.034,244.085,-65.303,-177.463,7.441,148.670
C00920=1166.029,244.333,-65.330,-177.461,7.443,148.670
C00921=1166.025,244.582,-65.357,-177.458,7.446,148.670
C00922=1166.020,244.831,-65.383,-177.455,7.449,148.670
C00923=1166.016,245.079,-65.410,-177.453,7.451,148.670
C00924=1166.012,245.327,-65.437,-177.450,7.454,148.669
C00925=1166.007,245.576,-65.464,-177.447,7.457,148.669
C00926=1166.002,245.824,-65.491,-177.444,7.459,148.669
C00927=1165.999,246.073,-65.517,-177.442,7.461,148.669
C00928=1165.994,246.322,-65.545,-177.439,7.464,148.669
C00929=1165.990,246.570,-65.572,-177.436,7.467,148.669
C00930=1165.985,246.819,-65.599,-177.434,7.469,148.669
C00931=1165.981,247.067,-65.625,-177.431,7.472,148.669
C00932=1165.977,247.315,-65.652,-177.428,7.475,148.668
C00933=1165.972,247.564,-65.679,-177.425,7.478,148.668
C00934=1165.967,247.812,-65.706,-177.423,7.480,148.668
C00935=1165.963,248.061,-65.733,-177.420,7.483,148.668
C00936=1165.959,248.309,-65.760,-177.418,7.486,148.668
C00937=1165.955,248.558,-65.787,-177.415,7.488,148.668
C00938=1165.950,248.807,-65.815,-177.412,7.491,148.668
C00939=1165.945,249.055,-65.842,-177.410,7.494,148.668
C00940=1165.941,249.304,-65.869,-177.407,7.497,148.668
C00941=1165.937,249.552,-65.895,-177.405,7.499,148.668
C00942=1165.932,249.801,-65.922,-177.402,7.502,148.667
C00943=1165.928,250.050,-65.950,-177.399,7.504,148.667
C00944=1165.924,250.298,-65.977,-177.396,7.507,148.667
C00945=1165.919,250.546,-66.004,-177.394,7.509,148.667
C00946=1165.914,250.795,-66.031,-177.391,7.512,148.667
C00947=1165.910,251.043,-66.059,-177.388,7.515,148.667
C00948=1165.906,251.291,-66.085,-177.385,7.518,148.667
C00949=1165.902,251.540,-66.113,-177.383,7.520,148.667
C00950=1165.897,251.788,-66.140,-177.380,7.523,148.666
C00951=1165.893,252.037,-66.167,-177.377,7.526,148.666
C00952=1165.888,252.285,-66.194,-177.374,7.529,148.666
C00953=1165.884,252.535,-66.222,-177.372,7.531,148.666
C00954=1165.880,252.782,-66.250,-177.370,7.534,148.666
C00955=1165.875,253.031,-66.277,-177.367,7.537,148.666
C00956=1165.870,253.279,-66.304,-177.364,7.540,148.666
C00957=1165.866,253.527,-66.331,-177.361,7.542,148.666
C00958=1165.862,253.776,-66.359,-177.359,7.545,148.666
C00959=1165.857,254.025,-66.386,-177.356,7.548,148.666
C00960=1165.853,254.273,-66.414,-177.353,7.551,148.666
C00961=1165.848,254.521,-66.441,-177.351,7.553,148.665
C00962=1165.844,254.771,-66.468,-177.348,7.556,148.665
C00963=1165.840,255.018,-66.496,-177.345,7.559,148.665
C00964=1165.835,255.267,-66.523,-177.343,7.562,148.665
C00965=1165.832,255.515,-66.551,-177.340,7.565,148.665
C00966=1165.827,255.764,-66.578,-177.338,7.567,148.665
C00967=1165.822,256.012,-66.606,-177.334,7.569,148.665
C00968=1165.818,256.260,-66.633,-177.332,7.572,148.665
C00969=1165.814,256.510,-66.661,-177.329,7.575,148.665
C00970=1165.809,256.757,-66.688,-177.327,7.577,148.665
C00971=1165.805,257.006,-66.715,-177.324,7.580,148.665
C00972=1165.801,257.254,-66.743,-177.321,7.583,148.664
C00973=1165.796,257.503,-66.771,-177.318,7.586,148.664
C00974=1165.791,257.751,-66.799,-177.316,7.589,148.664
C00975=1165.788,258.000,-66.827,-177.314,7.591,148.664
C00976=1165.783,258.248,-66.854,-177.311,7.594,148.664
C00977=1165.779,258.496,-66.882,-177.308,7.597,148.664
C00978=1165.774,258.745,-66.909,-177.305,7.600,148.664
C00979=1165.770,258.993,-66.937,-177.303,7.603,148.664
C00980=1165.765,259.242,-66.964,-177.300,7.605,148.664
C00981=1165.761,259.491,-66.993,-177.297,7.608,148.664
C00982=1165.757,259.738,-67.021,-177.294,7.611,148.664
C00983=1165.753,259.988,-67.048,-177.292,7.614,148.664
C00984=1165.748,260.236,-67.076,-177.289,7.617,148.664
C00985=1165.744,260.483,-67.104,-177.287,7.619,148.663
C00986=1165.739,260.733,-67.132,-177.284,7.622,148.663
C00987=1165.735,260.981,-67.159,-177.281,7.625,148.663
C00988=1165.731,261.229,-67.188,-177.278,7.628,148.663
C00989=1165.727,261.477,-67.215,-177.276,7.631,148.663
C00990=1165.722,261.751,-67.246,-177.273,7.634,148.663
C00991=1165.717,262.024,-67.277,-177.270,7.637,148.663
C00992=1165.712,262.297,-67.307,-177.267,7.640,148.663
C00993=1165.707,262.570,-67.338,-177.265,7.643,148.663
C00994=1165.703,262.819,-67.366,-177.262,7.645,148.663
C00995=1165.699,263.067,-67.394,-177.259,7.648,148.663
C00996=1165.694,263.315,-67.421,-177.256,7.651,148.663
C00997=1165.689,263.564,-67.450,-177.254,7.654,148.663
C00998=1165.685,263.812,-67.478,-177.251,7.657,148.663
C00999=1165.681,264.060,-67.506,-177.249,7.659,148.663
C01000=1165.676,264.309,-67.534,-177.246,7.662,148.663
C01001=1165.672,264.557,-67.562,-177.243,7.665,148.662
C01002=1165.668,264.805,-67.590,-177.240,7.668,148.662
C01003=1165.663,265.055,-67.618,-177.238,7.671,148.662
C01004=1165.659,265.302,-67.646,-177.235,7.674,148.662
C01005=1165.654,265.551,-67.675,-177.233,7.676,148.662
C01006=1165.650,265.799,-67.703,-177.230,7.679,148.662
C01007=1165.646,266.048,-67.731,-177.227,7.682,148.662
C01008=1165.641,266.296,-67.759,-177.224,7.685,148.662
C01009=1165.638,266.545,-67.787,-177.222,7.688,148.662
C01010=1165.632,266.793,-67.816,-177.219,7.691,148.662
C01011=1165.629,267.041,-67.844,-177.217,7.693,148.662
C01012=1165.624,267.290,-67.872,-177.214,7.696,148.662
C01013=1165.620,267.538,-67.900,-177.211,7.699,148.662
C01014=1165.615,267.786,-67.928,-177.208,7.702,148.662
C01015=1165.611,268.035,-67.957,-177.206,7.705,148.662
C01016=1165.607,268.282,-67.985,-177.203,7.708,148.662
C01017=1165.602,268.531,-68.014,-177.200,7.711,148.662
C01018=1165.598,268.779,-68.042,-177.198,7.713,148.661
C01019=1165.594,269.028,-68.071,-177.195,7.716,148.661
C01020=1165.590,269.276,-68.099,-177.193,7.719,148.661
C01021=1165.585,269.525,-68.127,-177.190,7.722,148.661
C01022=1165.581,269.773,-68.155,-177.187,7.725,148.661
C01023=1165.576,270.021,-68.184,-177.184,7.728,148.661
C01024=1165.573,270.269,-68.212,-177.181,7.731,148.661
C01025=1165.568,270.518,-68.241,-177.179,7.734,148.661
C01026=1165.563,270.766,-68.270,-177.177,7.736,148.661
C01027=1165.559,271.015,-68.298,-177.174,7.739,148.661
C01028=1165.554,271.262,-68.327,-177.172,7.742,148.661
C01029=1165.551,271.511,-68.355,-177.169,7.745,148.661
C01030=1165.546,271.760,-68.384,-177.166,7.748,148.661
C01031=1165.541,272.008,-68.412,-177.163,7.751,148.661
C01032=1165.538,272.256,-68.441,-177.160,7.754,148.661
C01033=1165.533,272.505,-68.470,-177.158,7.757,148.661
C01034=1165.529,272.753,-68.497,-177.156,7.759,148.661
C01035=1165.525,273.001,-68.527,-177.153,7.762,148.661
C01036=1165.520,273.249,-68.555,-177.150,7.765,148.661
C01037=1165.516,273.498,-68.583,-177.148,7.768,148.661
C01038=1165.512,273.746,-68.613,-177.145,7.771,148.661
C01039=1165.507,273.994,-68.641,-177.142,7.774,148.661
C01040=1165.503,274.242,-68.670,-177.139,7.777,148.661
C01041=1165.499,274.491,-68.699,-177.137,7.780,148.661
C01042=1165.494,274.740,-68.728,-177.134,7.783,148.661
C01043=1165.490,274.987,-68.756,-177.132,7.785,148.661
C01044=1165.486,275.236,-68.785,-177.129,7.788,148.661
C01045=1165.481,275.484,-68.814,-177.126,7.791,148.660
C01046=1165.476,275.733,-68.843,-177.124,7.795,148.661
C01047=1165.473,275.981,-68.871,-177.121,7.798,148.661
C01048=1165.468,276.229,-68.900,-177.119,7.801,148.661
C01049=1165.464,276.477,-68.929,-177.116,7.804,148.661
C01050=1165.460,276.726,-68.957,-177.113,7.807,148.660
C01051=1165.456,276.974,-68.987,-177.110,7.809,148.660
C01052=1165.451,277.223,-69.016,-177.107,7.812,148.660
C01053=1165.446,277.470,-69.045,-177.106,7.815,148.661
C01054=1165.442,277.719,-69.074,-177.103,7.818,148.660
C01055=1165.438,277.967,-69.102,-177.100,7.821,148.660
C01056=1165.434,278.215,-69.132,-177.098,7.824,148.660
C01057=1165.430,278.464,-69.160,-177.095,7.827,148.660
C01058=1165.425,278.712,-69.190,-177.092,7.830,148.660
C01059=1165.421,278.960,-69.219,-177.089,7.833,148.660
C01060=1165.416,279.209,-69.248,-177.087,7.836,148.660
C01061=1165.413,279.457,-69.277,-177.084,7.839,148.660
C01062=1165.408,279.705,-69.306,-177.081,7.842,148.660
C01063=1165.404,279.953,-69.335,-177.079,7.845,148.660
C01064=1165.399,280.202,-69.364,-177.076,7.848,148.660
C01065=1165.395,280.450,-69.393,-177.073,7.851,148.660
C01066=1165.391,280.698,-69.423,-177.071,7.853,148.660
C01067=1165.386,280.946,-69.452,-177.069,7.856,148.660
C01068=1165.382,281.195,-69.481,-177.066,7.859,148.660
C01069=1165.378,281.443,-69.510,-177.063,7.862,148.660
C01070=1165.374,281.691,-69.539,-177.060,7.865,148.660
C01071=1165.370,281.939,-69.568,-177.058,7.868,148.660
C01072=1165.366,282.188,-69.598,-177.055,7.871,148.660
C01073=1165.361,282.436,-69.626,-177.053,7.874,148.660
C01074=1165.357,282.684,-69.656,-177.050,7.877,148.660
C01075=1165.352,282.932,-69.685,-177.047,7.880,148.660
C01076=1165.348,283.180,-69.715,-177.045,7.884,148.660
C01077=1165.344,283.429,-69.744,-177.042,7.886,148.660
C01078=1165.340,283.677,-69.773,-177.039,7.889,148.660
C01079=1165.336,283.925,-69.803,-177.037,7.892,148.660
C01080=1165.331,284.173,-69.832,-177.034,7.895,148.660
C01081=1165.327,284.421,-69.861,-177.032,7.899,148.660
C01082=1165.322,284.669,-69.891,-177.029,7.902,148.660
C01083=1165.318,284.918,-69.920,-177.027,7.904,148.660
C01084=1165.313,285.167,-69.950,-177.024,7.907,148.660
C01085=1165.309,285.415,-69.979,-177.022,7.910,148.660
C01086=1165.305,285.663,-70.009,-177.019,7.913,148.660
C01087=1165.301,285.911,-70.039,-177.016,7.916,148.660
C01088=1165.297,286.159,-70.068,-177.013,7.919,148.660
C01089=1165.292,286.408,-70.098,-177.011,7.922,148.660
C01090=1165.288,286.656,-70.127,-177.008,7.925,148.660
C01091=1165.284,286.904,-70.157,-177.006,7.928,148.660
C01092=1165.279,287.152,-70.186,-177.003,7.931,148.660
C01093=1165.275,287.400,-70.215,-177.001,7.934,148.661
C01094=1165.270,287.675,-70.248,-176.998,7.937,148.660
C01095=1165.266,287.950,-70.281,-176.994,7.941,148.660
C01096=1165.261,288.225,-70.314,-176.992,7.944,148.660
C01097=1165.256,288.500,-70.347,-176.988,7.948,148.660
C01098=1165.252,288.749,-70.376,-176.986,7.951,148.661
C01099=1165.248,288.997,-70.406,-176.983,7.954,148.661
C01100=1165.244,289.244,-70.436,-176.981,7.957,148.661
C01101=1165.239,289.493,-70.466,-176.978,7.960,148.661
C01102=1165.235,289.741,-70.496,-176.976,7.963,148.661
C01103=1165.230,289.990,-70.525,-176.973,7.966,148.661
C01104=1165.227,290.237,-70.555,-176.970,7.969,148.661
C01105=1165.222,290.485,-70.585,-176.968,7.973,148.661
C01106=1165.217,290.734,-70.615,-176.965,7.976,148.661
C01107=1165.213,290.982,-70.644,-176.963,7.978,148.661
C01108=1165.209,291.230,-70.674,-176.960,7.981,148.661
C01109=1165.205,291.478,-70.704,-176.958,7.984,148.661
C01110=1165.200,291.727,-70.734,-176.955,7.987,148.661
C01111=1165.196,291.974,-70.764,-176.952,7.990,148.661
C01112=1165.192,292.223,-70.793,-176.950,7.993,148.661
C01113=1165.187,292.471,-70.823,-176.947,7.996,148.661
C01114=1165.183,292.719,-70.854,-176.945,7.999,148.661
C01115=1165.180,292.968,-70.883,-176.942,8.002,148.661
C01116=1165.175,293.216,-70.914,-176.939,8.005,148.661
C01117=1165.171,293.464,-70.944,-176.937,8.008,148.661
C01118=1165.167,293.712,-70.974,-176.934,8.012,148.661
C01119=1165.162,293.960,-71.004,-176.932,8.015,148.661
C01120=1165.158,294.208,-71.034,-176.929,8.018,148.661
C01121=1165.154,294.456,-71.064,-176.927,8.021,148.661
C01122=1165.150,294.704,-71.094,-176.924,8.024,148.661
C01123=1165.145,294.952,-71.124,-176.921,8.027,148.661
C01124=1165.141,295.200,-71.154,-176.919,8.030,148.661
C01125=1165.137,295.449,-71.184,-176.916,8.033,148.661
C01126=1165.133,295.697,-71.214,-176.913,8.037,148.661
C01127=1165.128,295.946,-71.245,-176.910,8.040,148.662
C01128=1165.125,296.193,-71.275,-176.908,8.043,148.662
C01129=1165.120,296.442,-71.305,-176.905,8.046,148.661
C01130=1165.116,296.690,-71.335,-176.903,8.049,148.662
C01131=1165.112,296.937,-71.365,-176.900,8.052,148.662
C01132=1165.108,297.186,-71.395,-176.897,8.055,148.662
C01133=1165.104,297.434,-71.426,-176.895,8.059,148.662
C01134=1165.099,297.682,-71.456,-176.892,8.062,148.662
C01135=1165.095,297.930,-71.486,-176.889,8.065,148.662
C01136=1165.090,298.178,-71.517,-176.887,8.068,148.662
C01137=1165.086,298.426,-71.547,-176.884,8.071,148.662
C01138=1165.082,298.675,-71.577,-176.882,8.074,148.662
C01139=1165.078,298.923,-71.608,-176.879,8.077,148.662
C01140=1165.074,299.171,-71.638,-176.877,8.080,148.662
C01141=1165.069,299.419,-71.669,-176.874,8.083,148.662
C01142=1165.065,299.667,-71.698,-176.872,8.086,148.662
C01143=1165.061,299.916,-71.730,-176.869,8.090,148.662
C01144=1165.057,300.163,-71.760,-176.867,8.093,148.662
C01145=1165.052,300.411,-71.790,-176.864,8.095,148.662
C01146=1165.048,300.659,-71.821,-176.861,8.099,148.662
C01147=1165.044,300.908,-71.852,-176.859,8.102,148.662
C01148=1165.040,301.156,-71.882,-176.856,8.105,148.663
C01149=1165.036,301.404,-71.912,-176.854,8.108,148.663
C01150=1165.031,301.652,-71.943,-176.851,8.111,148.663
C01151=1165.027,301.900,-71.974,-176.849,8.114,148.663
C01152=1165.023,302.148,-72.004,-176.846,8.117,148.663
C01153=1165.019,302.396,-72.035,-176.844,8.121,148.663
C01154=1165.014,302.644,-72.066,-176.841,8.124,148.663
C01155=1165.011,302.892,-72.096,-176.838,8.126,148.663
C01156=1165.006,303.140,-72.127,-176.835,8.131,148.663
C01157=1165.001,303.388,-72.158,-176.833,8.134,148.663
C01158=1164.998,303.636,-72.188,-176.830,8.137,148.663
C01159=1164.994,303.885,-72.219,-176.827,8.140,148.663
C01160=1164.989,304.133,-72.250,-176.825,8.143,148.663
C01161=1164.984,304.380,-72.280,-176.822,8.146,148.663
C01162=1164.981,304.629,-72.311,-176.820,8.149,148.664
C01163=1164.976,304.877,-72.342,-176.817,8.152,148.664
C01164=1164.972,305.125,-72.372,-176.815,8.155,148.664
C01165=1164.968,305.373,-72.404,-176.812,8.159,148.664
C01166=1164.964,305.621,-72.434,-176.810,8.162,148.664
C01167=1164.959,305.869,-72.465,-176.807,8.165,148.664
C01168=1164.955,306.118,-72.496,-176.805,8.168,148.664
C01169=1164.951,306.366,-72.526,-176.802,8.171,148.664
C01170=1164.947,306.613,-72.557,-176.800,8.174,148.664
C01171=1164.943,306.861,-72.588,-176.797,8.177,148.664
C01172=1164.938,307.109,-72.619,-176.794,8.181,148.664
C01173=1164.934,307.357,-72.650,-176.792,8.184,148.664
C01174=1164.930,307.606,-72.681,-176.789,8.187,148.664
C01175=1164.925,307.854,-72.712,-176.787,8.191,148.665
C01176=1164.922,308.102,-72.744,-176.784,8.194,148.665
C01177=1164.918,308.350,-72.774,-176.782,8.197,148.665
C01178=1164.913,308.597,-72.805,-176.779,8.200,148.665
C01179=1164.909,308.846,-72.836,-176.776,8.203,148.665
C01180=1164.905,309.093,-72.867,-176.774,8.206,148.665
C01181=1164.901,309.342,-72.898,-176.771,8.210,148.665
C01182=1164.896,309.590,-72.929,-176.769,8.212,148.665
C01183=1164.892,309.837,-72.961,-176.766,8.216,148.665
C01184=1164.888,310.086,-72.992,-176.763,8.220,148.665
C01185=1164.883,310.334,-73.023,-176.761,8.223,148.665
C01186=1164.879,310.582,-73.054,-176.758,8.226,148.665
C01187=1164.876,310.830,-73.085,-176.756,8.229,148.666
C01188=1164.872,311.078,-73.116,-176.753,8.232,148.666
C01189=1164.867,311.326,-73.147,-176.751,8.235,148.666
C01190=1164.863,311.574,-73.178,-176.748,8.238,148.666
C01191=1164.859,311.822,-73.210,-176.746,8.242,148.666
C01192=1164.854,312.070,-73.241,-176.743,8.245,148.666
C01193=1164.851,312.318,-73.272,-176.741,8.248,148.666
C01194=1164.846,312.566,-73.303,-176.737,8.252,148.666
C01195=1164.842,312.814,-73.335,-176.735,8.255,148.666
C01196=1164.838,313.062,-73.366,-176.733,8.258,148.667
C01197=1164.834,313.310,-73.398,-176.730,8.261,148.667
C01198=1164.829,313.587,-73.432,-176.728,8.265,148.667
C01199=1164.824,313.864,-73.467,-176.724,8.268,148.667
C01200=1164.820,314.142,-73.503,-176.722,8.272,148.667
C01201=1164.815,314.418,-73.538,-176.719,8.275,148.667
C01202=1164.811,314.667,-73.569,-176.716,8.279,148.667
C01203=1164.806,314.914,-73.601,-176.714,8.282,148.667
C01204=1164.803,315.162,-73.633,-176.711,8.286,148.667
C01205=1164.798,315.410,-73.663,-176.708,8.289,148.667
C01206=1164.794,315.658,-73.695,-176.706,8.292,148.668
C01207=1164.790,315.906,-73.727,-176.704,8.295,148.668
C01208=1164.786,316.154,-73.758,-176.701,8.298,148.668
C01209=1164.782,316.402,-73.789,-176.699,8.302,148.668
C01210=1164.777,316.650,-73.822,-176.696,8.305,148.668
C01211=1164.773,316.899,-73.853,-176.693,8.308,148.668
C01212=1164.769,317.146,-73.884,-176.690,8.312,148.668
C01213=1164.765,317.394,-73.916,-176.688,8.315,148.668
C01214=1164.761,317.641,-73.948,-176.686,8.318,148.668
C01215=1164.757,317.890,-73.979,-176.683,8.321,148.668
C01216=1164.752,318.138,-74.011,-176.681,8.325,148.669
C01217=1164.748,318.386,-74.043,-176.678,8.328,148.669
C01218=1164.744,318.634,-74.075,-176.676,8.331,148.669
C01219=1164.740,318.881,-74.106,-176.673,8.335,148.669
C01220=1164.735,319.130,-74.138,-176.670,8.338,148.669
C01221=1164.732,319.378,-74.170,-176.668,8.341,148.669
C01222=1164.727,319.625,-74.201,-176.665,8.344,148.669
C01223=1164.724,319.874,-74.233,-176.663,8.347,148.669
C01224=1164.719,320.122,-74.265,-176.660,8.351,148.670
C01225=1164.715,320.369,-74.297,-176.658,8.354,148.670
C01226=1164.711,320.617,-74.329,-176.655,8.358,148.670
C01227=1164.707,320.865,-74.361,-176.652,8.361,148.670
C01228=1164.702,321.113,-74.393,-176.650,8.364,148.670
C01229=1164.699,321.361,-74.425,-176.647,8.367,148.670
C01230=1164.695,321.609,-74.456,-176.645,8.371,148.670
C01231=1164.690,321.857,-74.488,-176.642,8.374,148.670
C01232=1164.686,322.105,-74.520,-176.640,8.377,148.671
C01233=1164.683,322.353,-74.552,-176.637,8.381,148.671
C01234=1164.678,322.600,-74.584,-176.634,8.384,148.671
C01235=1164.674,322.848,-74.616,-176.632,8.387,148.671
C01236=1164.670,323.096,-74.648,-176.630,8.391,148.671
C01237=1164.666,323.345,-74.680,-176.628,8.394,148.671
C01238=1164.661,323.592,-74.712,-176.625,8.397,148.671
C01239=1164.658,323.840,-74.744,-176.622,8.401,148.672
C01240=1164.653,324.089,-74.776,-176.620,8.404,148.672
C01241=1164.649,324.336,-74.808,-176.617,8.407,148.672
C01242=1164.645,324.584,-74.841,-176.615,8.411,148.672
C01243=1164.641,324.832,-74.873,-176.612,8.414,148.672
C01244=1164.637,325.080,-74.905,-176.610,8.417,148.672
C01245=1164.633,325.328,-74.937,-176.607,8.421,148.673
C01246=1164.629,325.575,-74.968,-176.604,8.424,148.673
C01247=1164.624,325.824,-75.001,-176.602,8.427,148.673
C01248=1164.621,326.071,-75.033,-176.599,8.430,148.673
C01249=1164.616,326.320,-75.066,-176.597,8.434,148.673
C01250=1164.612,326.567,-75.097,-176.594,8.438,148.673
C01251=1164.608,326.815,-75.130,-176.591,8.441,148.673
C01252=1164.604,327.063,-75.162,-176.589,8.444,148.674
C01253=1164.600,327.311,-75.195,-176.587,8.447,148.674
C01254=1164.596,327.559,-75.227,-176.585,8.451,148.674
C01255=1164.591,327.806,-75.259,-176.581,8.454,148.674
C01256=1164.588,328.054,-75.291,-176.579,8.458,148.674
C01257=1164.583,328.302,-75.324,-176.577,8.461,148.674
C01258=1164.579,328.550,-75.357,-176.574,8.464,148.675
C01259=1164.575,328.798,-75.389,-176.572,8.467,148.675
C01260=1164.570,329.046,-75.421,-176.569,8.471,148.675
C01261=1164.567,329.293,-75.453,-176.566,8.475,148.675
C01262=1164.562,329.542,-75.486,-176.564,8.478,148.675
C01263=1164.558,329.789,-75.519,-176.561,8.481,148.675
C01264=1164.555,330.037,-75.551,-176.559,8.484,148.675
C01265=1164.550,330.285,-75.584,-176.556,8.488,148.676
C01266=1164.547,330.533,-75.616,-176.554,8.492,148.676
C01267=1164.542,330.780,-75.649,-176.552,8.495,148.676
C01268=1164.537,331.029,-75.681,-176.549,8.498,148.676
C01269=1164.534,331.276,-75.714,-176.547,8.501,148.676
C01270=1164.530,331.524,-75.746,-176.544,8.505,148.676
C01271=1164.526,331.772,-75.779,-176.541,8.509,148.677
C01272=1164.522,332.020,-75.811,-176.539,8.512,148.677
C01273=1164.518,332.268,-75.844,-176.536,8.515,148.677
C01274=1164.513,332.516,-75.877,-176.534,8.518,148.677
C01275=1164.508,332.763,-75.909,-176.531,8.522,148.677
C01276=1164.505,333.011,-75.942,-176.529,8.526,148.678
C01277=1164.501,333.259,-75.974,-176.527,8.529,148.678
C01278=1164.496,333.507,-76.008,-176.524,8.532,148.678
C01279=1164.492,333.754,-76.041,-176.521,8.536,148.678
C01280=1164.489,334.002,-76.073,-176.519,8.539,148.678
C01281=1164.485,334.250,-76.106,-176.516,8.543,148.678
C01282=1164.480,334.498,-76.139,-176.514,8.546,148.679
C01283=1164.476,334.746,-76.171,-176.512,8.549,148.679
C01284=1164.473,334.994,-76.204,-176.509,8.553,148.679
C01285=1164.468,335.241,-76.237,-176.506,8.556,148.679
C01286=1164.464,335.489,-76.270,-176.504,8.560,148.679
C01287=1164.460,335.737,-76.303,-176.502,8.563,148.679
C01288=1164.456,335.985,-76.336,-176.499,8.567,148.680
C01289=1164.452,336.233,-76.368,-176.497,8.570,148.680
C01290=1164.448,336.480,-76.401,-176.494,8.574,148.680
C01291=1164.444,336.728,-76.435,-176.492,8.577,148.680
C01292=1164.440,336.976,-76.467,-176.489,8.581,148.681
C01293=1164.435,337.224,-76.500,-176.486,8.584,148.681
C01294=1164.431,337.472,-76.533,-176.484,8.587,148.681
C01295=1164.427,337.720,-76.567,-176.482,8.591,148.681
C01296=1164.423,337.967,-76.600,-176.479,8.595,148.681
C01297=1164.420,338.215,-76.632,-176.477,8.598,148.681
C01298=1164.415,338.462,-76.665,-176.474,8.601,148.682
C01299=1164.411,338.710,-76.699,-176.472,8.604,148.682
C01300=1164.407,338.958,-76.732,-176.469,8.609,148.682
C01301=1164.403,339.206,-76.765,-176.467,8.612,148.682
C01302=1164.398,339.486,-76.802,-176.464,8.616,148.683
C01303=1164.394,339.765,-76.839,-176.461,8.620,148.683
C01304=1164.389,340.045,-76.877,-176.458,8.623,148.683
C01305=1164.384,340.325,-76.914,-176.455,8.627,148.683
C01306=1164.380,340.572,-76.947,-176.453,8.631,148.683
C01307=1164.376,340.820,-76.981,-176.450,8.635,148.684
C01308=1164.372,341.068,-77.014,-176.448,8.638,148.684
C01309=1164.368,341.316,-77.047,-176.446,8.641,148.684
C01310=1164.364,341.563,-77.080,-176.443,8.645,148.684
C01311=1164.360,341.810,-77.114,-176.441,8.649,148.684
C01312=1164.356,342.058,-77.147,-176.438,8.652,148.685
C01313=1164.352,342.307,-77.181,-176.436,8.655,148.685
C01314=1164.348,342.554,-77.214,-176.433,8.659,148.685
C01315=1164.344,342.802,-77.247,-176.431,8.663,148.685
C01316=1164.340,343.050,-77.280,-176.428,8.666,148.686
C01317=1164.336,343.297,-77.313,-176.426,8.670,148.686
C01318=1164.331,343.545,-77.348,-176.423,8.673,148.686
C01319=1164.327,343.793,-77.381,-176.421,8.677,148.686
C01320=1164.323,344.040,-77.414,-176.418,8.681,148.686
C01321=1164.319,344.289,-77.448,-176.416,8.684,148.687
C01322=1164.315,344.536,-77.481,-176.414,8.687,148.687
C01323=1164.311,344.784,-77.515,-176.411,8.691,148.687
C01324=1164.307,345.031,-77.548,-176.408,8.695,148.687
C01325=1164.302,345.279,-77.581,-176.406,8.698,148.688
C01326=1164.298,345.526,-77.615,-176.404,8.701,148.688
C01327=1164.295,345.775,-77.649,-176.401,8.705,148.688
C01328=1164.291,346.023,-77.682,-176.399,8.709,148.688
C01329=1164.287,346.270,-77.716,-176.396,8.712,148.688
C01330=1164.283,346.517,-77.749,-176.393,8.716,148.689
C01331=1164.278,346.765,-77.783,-176.392,8.720,148.689
C01332=1164.275,347.013,-77.817,-176.389,8.723,148.689
C01333=1164.271,347.261,-77.850,-176.386,8.727,148.690
C01334=1164.267,347.508,-77.884,-176.384,8.730,148.690
C01335=1164.262,347.756,-77.918,-176.382,8.734,148.690
C01336=1164.258,348.003,-77.952,-176.379,8.738,148.690
C01337=1164.254,348.252,-77.985,-176.377,8.741,148.691
C01338=1164.251,348.499,-78.019,-176.374,8.744,148.691
C01339=1164.246,348.747,-78.053,-176.372,8.748,148.691
C01340=1164.242,348.994,-78.087,-176.369,8.752,148.691
C01341=1164.238,349.242,-78.120,-176.367,8.755,148.691
C01342=1164.234,349.490,-78.155,-176.364,8.759,148.692
C01343=1164.230,349.738,-78.188,-176.362,8.763,148.692
C01344=1164.226,349.985,-78.222,-176.360,8.766,148.692
C01345=1164.222,350.233,-78.256,-176.357,8.770,148.693
C01346=1164.218,350.481,-78.290,-176.355,8.773,148.693
C01347=1164.214,350.728,-78.324,-176.352,8.777,148.693
C01348=1164.210,350.976,-78.358,-176.350,8.781,148.693
C01349=1164.206,351.223,-78.392,-176.348,8.784,148.694
C01350=1164.202,351.471,-78.425,-176.345,8.788,148.694
C01351=1164.198,351.719,-78.460,-176.343,8.792,148.694
C01352=1164.194,351.966,-78.493,-176.340,8.795,148.694
C01353=1164.190,352.214,-78.527,-176.338,8.798,148.695
C01354=1164.186,352.462,-78.561,-176.335,8.803,148.695
C01355=1164.182,352.709,-78.595,-176.333,8.806,148.695
C01356=1164.177,352.957,-78.630,-176.331,8.809,148.695
C01357=1164.174,353.205,-78.664,-176.328,8.814,148.696
C01358=1164.169,353.453,-78.698,-176.326,8.817,148.696
C01359=1164.165,353.700,-78.732,-176.323,8.821,148.696
C01360=1164.162,353.948,-78.766,-176.321,8.825,148.697
C01361=1164.158,354.195,-78.800,-176.319,8.828,148.697
C01362=1164.154,354.442,-78.834,-176.316,8.832,148.697
C01363=1164.149,354.691,-78.868,-176.314,8.835,148.697
C01364=1164.146,354.938,-78.902,-176.312,8.839,148.698
C01365=1164.141,355.185,-78.937,-176.309,8.843,148.698
C01366=1164.138,355.433,-78.971,-176.307,8.846,148.698
C01367=1164.133,355.681,-79.005,-176.304,8.850,148.698
C01368=1164.130,355.928,-79.040,-176.302,8.854,148.699
C01369=1164.125,356.176,-79.074,-176.299,8.857,148.699
C01370=1164.122,356.424,-79.109,-176.297,8.861,148.699
C01371=1164.118,356.671,-79.143,-176.294,8.865,148.700
C01372=1164.113,356.918,-79.177,-176.292,8.869,148.700
C01373=1164.110,357.166,-79.211,-176.290,8.872,148.700
C01374=1164.105,357.414,-79.246,-176.287,8.876,148.701
C01375=1164.102,357.662,-79.280,-176.285,8.880,148.701
C01376=1164.098,357.909,-79.315,-176.283,8.883,148.701
C01377=1164.094,358.157,-79.349,-176.280,8.887,148.701
C01378=1164.090,358.404,-79.383,-176.278,8.891,148.702
C01379=1164.086,358.652,-79.418,-176.276,8.894,148.702
C01380=1164.082,358.899,-79.452,-176.273,8.899,148.702
C01381=1164.077,359.147,-79.486,-176.271,8.902,148.703
C01382=1164.073,359.395,-79.521,-176.268,8.906,148.703
C01383=1164.070,359.642,-79.555,-176.266,8.910,148.703
C01384=1164.066,359.890,-79.590,-176.263,8.914,148.704
C01385=1164.061,360.137,-79.625,-176.261,8.917,148.704
C01386=1164.058,360.385,-79.659,-176.258,8.921,148.704
C01387=1164.054,360.632,-79.694,-176.256,8.925,148.705
C01388=1164.050,360.880,-79.729,-176.254,8.928,148.705
C01389=1164.046,361.127,-79.763,-176.251,8.933,148.705
C01390=1164.042,361.375,-79.798,-176.249,8.936,148.706
C01391=1164.038,361.623,-79.833,-176.246,8.940,148.706
C01392=1164.034,361.870,-79.867,-176.244,8.944,148.706
C01393=1164.030,362.118,-79.902,-176.242,8.948,148.707
C01394=1164.026,362.365,-79.937,-176.240,8.951,148.707
C01395=1164.022,362.613,-79.972,-176.237,8.955,148.707
C01396=1164.018,362.860,-80.006,-176.235,8.959,148.708
C01397=1164.014,363.108,-80.040,-176.233,8.962,148.708
C01398=1164.010,363.355,-80.076,-176.230,8.967,148.708
C01399=1164.006,363.603,-80.110,-176.228,8.970,148.709
C01400=1164.002,363.851,-80.146,-176.225,8.974,148.709
C01401=1163.999,364.098,-80.180,-176.224,8.978,148.709
C01402=1163.995,364.346,-80.215,-176.221,8.982,148.710
C01403=1163.990,364.593,-80.250,-176.219,8.986,148.710
C01404=1163.986,364.841,-80.285,-176.217,8.989,148.710
C01405=1163.983,365.089,-80.320,-176.214,8.994,148.711
C01406=1163.978,365.371,-80.360,-176.212,8.998,148.711
C01407=1163.974,365.654,-80.399,-176.209,9.002,148.712
C01408=1163.969,365.935,-80.439,-176.206,9.006,148.712
C01409=1163.964,366.218,-80.479,-176.204,9.011,148.713
C01410=1163.961,366.465,-80.514,-176.202,9.014,148.713
C01411=1163.957,366.713,-80.549,-176.200,9.019,148.713
C01412=1163.953,366.960,-80.584,-176.198,9.023,148.714
C01413=1163.949,367.208,-80.619,-176.195,9.026,148.714
C01414=1163.945,367.456,-80.654,-176.193,9.030,148.715
C01415=1163.941,367.703,-80.690,-176.191,9.034,148.715
C01416=1163.937,367.951,-80.724,-176.189,9.038,148.716
C01417=1163.933,368.198,-80.760,-176.187,9.042,148.716
C01418=1163.929,368.446,-80.794,-176.185,9.045,148.716
C01419=1163.925,368.693,-80.830,-176.183,9.050,148.717
C01420=1163.921,368.941,-80.865,-176.181,9.053,148.717
C01421=1163.917,369.188,-80.900,-176.179,9.057,148.718
C01422=1163.913,369.436,-80.935,-176.177,9.061,148.718
C01423=1163.909,369.683,-80.971,-176.175,9.065,148.719
C01424=1163.905,369.931,-81.006,-176.173,9.069,148.719
C01425=1163.901,370.178,-81.041,-176.171,9.072,148.719
C01426=1163.898,370.426,-81.077,-176.168,9.077,148.720
C01427=1163.893,370.672,-81.112,-176.167,9.081,148.721
C01428=1163.889,370.920,-81.147,-176.165,9.084,148.721
C01429=1163.886,371.168,-81.182,-176.163,9.088,148.721
C01430=1163.882,371.415,-81.218,-176.161,9.091,148.722
C01431=1163.878,371.662,-81.253,-176.159,9.096,148.722
C01432=1163.874,371.910,-81.288,-176.157,9.100,148.723
C01433=1163.870,372.158,-81.323,-176.156,9.103,148.723
C01434=1163.866,372.405,-81.359,-176.154,9.107,148.724
C01435=1163.861,372.653,-81.395,-176.152,9.111,148.724
C01436=1163.858,372.900,-81.430,-176.150,9.114,148.725
C01437=1163.854,373.148,-81.466,-176.148,9.119,148.725
C01438=1163.850,373.395,-81.501,-176.147,9.123,148.726
C01439=1163.846,373.642,-81.536,-176.145,9.127,148.727
C01440=1163.842,373.890,-81.571,-176.143,9.130,148.727
C01441=1163.839,374.137,-81.607,-176.142,9.134,148.728
C01442=1163.835,374.385,-81.642,-176.140,9.138,148.728
C01443=1163.830,374.633,-81.678,-176.139,9.142,148.729
C01444=1163.826,374.880,-81.714,-176.137,9.146,148.729
C01445=1163.823,375.127,-81.749,-176.136,9.149,148.730
C01446=1163.819,375.375,-81.785,-176.134,9.153,148.730
C01447=1163.815,375.622,-81.820,-176.132,9.157,148.731
C01448=1163.812,375.870,-81.856,-176.131,9.161,148.732
C01449=1163.807,376.117,-81.892,-176.129,9.165,148.732
C01450=1163.803,376.364,-81.927,-176.128,9.169,148.733
C01451=1163.799,376.612,-81.963,-176.127,9.173,148.733
C01452=1163.796,376.859,-81.998,-176.125,9.175,148.734
C01453=1163.792,377.107,-82.034,-176.124,9.179,148.734
C01454=1163.787,377.354,-82.070,-176.122,9.183,148.735
C01455=1163.783,377.601,-82.105,-176.121,9.187,148.736
C01456=1163.780,377.849,-82.141,-176.120,9.191,148.736
C01457=1163.776,378.096,-82.177,-176.119,9.195,148.737
C01458=1163.772,378.343,-82.213,-176.118,9.198,148.738
C01459=1163.768,378.591,-82.249,-176.116,9.202,148.738
C01460=1163.764,378.838,-82.284,-176.115,9.206,148.739
C01461=1163.759,379.086,-82.320,-176.114,9.209,148.740
C01462=1163.756,379.333,-82.356,-176.113,9.213,148.740
C01463=1163.752,379.581,-82.391,-176.112,9.217,148.741
C01464=1163.749,379.827,-82.427,-176.111,9.220,148.742
C01465=1163.744,380.075,-82.463,-176.109,9.224,148.742
C01466=1163.741,380.323,-82.499,-176.109,9.228,148.743
C01467=1163.737,380.570,-82.535,-176.107,9.232,148.744
C01468=1163.732,380.817,-82.570,-176.106,9.236,148.744
C01469=1163.729,381.064,-82.607,-176.105,9.239,148.745
C01470=1163.725,381.312,-82.642,-176.105,9.242,148.746
C01471=1163.721,381.560,-82.678,-176.104,9.246,148.746
C01472=1163.717,381.807,-82.714,-176.103,9.250,148.747
C01473=1163.714,382.054,-82.750,-176.102,9.253,148.748
C01474=1163.709,382.302,-82.786,-176.101,9.257,148.749
C01475=1163.706,382.549,-82.822,-176.100,9.260,148.749
C01476=1163.701,382.797,-82.858,-176.099,9.264,148.750
C01477=1163.698,383.044,-82.894,-176.099,9.268,148.751
C01478=1163.694,383.291,-82.929,-176.099,9.271,148.751
C01479=1163.689,383.539,-82.966,-176.098,9.274,148.752
C01480=1163.686,383.785,-83.002,-176.097,9.278,148.753
C01481=1163.682,384.033,-83.037,-176.096,9.282,148.754
C01482=1163.678,384.281,-83.074,-176.096,9.285,148.754
C01483=1163.674,384.528,-83.110,-176.095,9.288,148.755
C01484=1163.670,384.775,-83.146,-176.095,9.291,148.756
C01485=1163.666,385.023,-83.181,-176.094,9.295,148.757
C01486=1163.662,385.270,-83.218,-176.094,9.298,148.757
C01487=1163.659,385.518,-83.254,-176.093,9.302,148.758
C01488=1163.655,385.765,-83.289,-176.093,9.305,148.759
C01489=1163.651,386.012,-83.326,-176.092,9.308,148.760
C01490=1163.647,386.260,-83.362,-176.092,9.312,148.760
C01491=1163.643,386.507,-83.399,-176.092,9.315,148.761
C01492=1163.639,386.755,-83.434,-176.092,9.318,148.762
C01493=1163.635,387.002,-83.470,-176.092,9.321,148.763
C01494=1163.632,387.249,-83.507,-176.091,9.325,148.764
C01495=1163.628,387.497,-83.542,-176.091,9.327,148.764
C01496=1163.623,387.743,-83.579,-176.091,9.331,148.765
C01497=1163.620,387.991,-83.614,-176.090,9.334,148.766
C01498=1163.615,388.238,-83.651,-176.091,9.337,148.767
C01499=1163.612,388.485,-83.687,-176.091,9.340,148.767
C01500=1163.608,388.733,-83.723,-176.091,9.343,148.768
C01501=1163.604,388.980,-83.759,-176.090,9.346,148.769
C01502=1163.600,389.227,-83.796,-176.090,9.349,148.770
C01503=1163.596,389.475,-83.831,-176.090,9.353,148.771
C01504=1163.592,389.722,-83.868,-176.091,9.355,148.771
C01505=1163.589,389.969,-83.904,-176.091,9.358,148.772
C01506=1163.584,390.217,-83.941,-176.091,9.361,148.773
C01507=1163.581,390.464,-83.976,-176.091,9.364,148.774
C01508=1163.577,390.711,-84.013,-176.091,9.367,148.774
C01509=1163.573,390.959,-84.049,-176.091,9.369,148.775
C01510=1163.569,391.245,-84.090,-176.091,9.373,148.776
C01511=1163.564,391.530,-84.133,-176.091,9.377,148.777
C01512=1163.560,391.816,-84.174,-176.092,9.379,148.778
C01513=1163.555,392.100,-84.216,-176.092,9.382,148.779
C01514=1163.551,392.348,-84.252,-176.092,9.386,148.780
C01515=1163.547,392.595,-84.288,-176.092,9.389,148.781
C01516=1163.543,392.843,-84.324,-176.093,9.391,148.781
C01517=1163.540,393.090,-84.361,-176.093,9.394,148.782
C01518=1163.536,393.337,-84.398,-176.093,9.397,148.783
C01519=1163.532,393.584,-84.433,-176.093,9.399,148.784
C01520=1163.528,393.832,-84.470,-176.094,9.401,148.784
C01521=1163.525,394.080,-84.506,-176.095,9.404,148.785
C01522=1163.521,394.327,-84.543,-176.095,9.406,148.786
C01523=1163.516,394.575,-84.579,-176.095,9.409,148.787
C01524=1163.513,394.822,-84.615,-176.095,9.412,148.788
C01525=1163.509,395.069,-84.652,-176.096,9.414,148.788
C01526=1163.505,395.316,-84.688,-176.096,9.417,148.789
C01527=1163.501,395.563,-84.724,-176.097,9.419,148.790
C01528=1163.497,395.811,-84.760,-176.097,9.422,148.790
C01529=1163.493,396.058,-84.797,-176.098,9.424,148.791
C01530=1163.490,396.306,-84.832,-176.098,9.427,148.792
C01531=1163.486,396.553,-84.869,-176.098,9.429,148.793
C01532=1163.482,396.800,-84.906,-176.099,9.432,148.794
C01533=1163.478,397.047,-84.942,-176.099,9.434,148.794
C01534=1163.474,397.295,-84.978,-176.100,9.436,148.795
C01535=1163.470,397.542,-85.014,-176.100,9.439,148.796
C01536=1163.466,397.789,-85.051,-176.100,9.441,148.797
C01537=1163.463,398.036,-85.087,-176.101,9.443,148.797
C01538=1163.458,398.284,-85.123,-176.102,9.446,148.798
C01539=1163.454,398.531,-85.160,-176.102,9.448,148.799
C01540=1163.451,398.778,-85.196,-176.103,9.450,148.800
C01541=1163.446,399.026,-85.233,-176.103,9.452,148.800
C01542=1163.443,399.273,-85.269,-176.104,9.455,148.801
C01543=1163.439,399.521,-85.305,-176.105,9.457,148.802
C01544=1163.435,399.767,-85.341,-176.105,9.459,148.802
C01545=1163.431,400.015,-85.378,-176.105,9.461,148.803
C01546=1163.427,400.262,-85.414,-176.106,9.464,148.804
C01547=1163.423,400.509,-85.450,-176.107,9.466,148.805
C01548=1163.419,400.757,-85.487,-176.107,9.468,148.805
C01549=1163.416,401.004,-85.523,-176.108,9.470,148.806
C01550=1163.412,401.251,-85.560,-176.108,9.473,148.807
C01551=1163.407,401.498,-85.597,-176.109,9.475,148.808
C01552=1163.404,401.746,-85.632,-176.110,9.476,148.808
C01553=1163.400,401.993,-85.669,-176.110,9.479,148.809
C01554=1163.396,402.241,-85.705,-176.110,9.481,148.810
C01555=1163.392,402.488,-85.741,-176.110,9.483,148.810
C01556=1163.388,402.735,-85.778,-176.111,9.485,148.811
C01557=1163.384,402.983,-85.814,-176.112,9.487,148.812
C01558=1163.381,403.230,-85.851,-176.112,9.490,148.813
C01559=1163.377,403.477,-85.887,-176.113,9.491,148.813
C01560=1163.373,403.725,-85.923,-176.114,9.493,148.814
C01561=1163.369,403.972,-85.960,-176.115,9.495,148.814
C01562=1163.366,404.219,-85.997,-176.115,9.497,148.815
C01563=1163.361,404.467,-86.033,-176.115,9.499,148.816
C01564=1163.358,404.714,-86.069,-176.116,9.501,148.816
C01565=1163.354,404.961,-86.106,-176.116,9.503,148.817
C01566=1163.350,405.208,-86.143,-176.117,9.505,148.818
C01567=1163.346,405.456,-86.178,-176.118,9.507,148.818
C01568=1163.342,405.703,-86.215,-176.118,9.509,148.819
C01569=1163.338,405.950,-86.251,-176.118,9.511,148.820
C01570=1163.334,406.198,-86.288,-176.119,9.513,148.820
C01571=1163.330,406.445,-86.324,-176.120,9.515,148.821
C01572=1163.327,406.692,-86.361,-176.121,9.516,148.822
C01573=1163.322,406.939,-86.397,-176.121,9.519,148.822
C01574=1163.318,407.187,-86.434,-176.121,9.521,148.823
C01575=1163.315,407.434,-86.470,-176.122,9.523,148.824
C01576=1163.310,407.681,-86.506,-176.123,9.524,148.824
C01577=1163.308,407.929,-86.543,-176.123,9.526,148.825
C01578=1163.303,408.176,-86.580,-176.123,9.528,148.826
C01579=1163.299,408.423,-86.616,-176.124,9.530,148.826
C01580=1163.296,408.671,-86.652,-176.125,9.532,148.827
C01581=1163.292,408.918,-86.689,-176.125,9.533,148.828
C01582=1163.288,409.165,-86.725,-176.126,9.535,148.828
C01583=1163.284,409.413,-86.761,-176.126,9.538,148.829
C01584=1163.280,409.660,-86.798,-176.126,9.539,148.829
C01585=1163.276,409.907,-86.834,-176.127,9.541,148.830
C01586=1163.272,410.155,-86.870,-176.128,9.543,148.831
C01587=1163.268,410.402,-86.907,-176.129,9.544,148.831
C01588=1163.265,410.649,-86.944,-176.129,9.546,148.832
C01589=1163.260,410.896,-86.980,-176.129,9.548,148.832
C01590=1163.256,411.144,-87.017,-176.130,9.550,148.833
C01591=1163.253,411.391,-87.053,-176.130,9.552,148.834
C01592=1163.249,411.638,-87.090,-176.131,9.553,148.834
C01593=1163.246,411.885,-87.126,-176.131,9.555,148.835
C01594=1163.241,412.133,-87.162,-176.131,9.558,148.836
C01595=1163.237,412.380,-87.199,-176.132,9.559,148.836
C01596=1163.234,412.627,-87.236,-176.132,9.561,148.837
C01597=1163.230,412.875,-87.272,-176.133,9.563,148.837
C01598=1163.226,413.122,-87.309,-176.134,9.564,148.838
C01599=1163.222,413.369,-87.345,-176.134,9.566,148.838
C01600=1163.218,413.616,-87.382,-176.134,9.568,148.839
C01601=1163.214,413.864,-87.418,-176.135,9.570,148.840
C01602=1163.210,414.111,-87.454,-176.135,9.572,148.840
C01603=1163.206,414.358,-87.491,-176.136,9.573,148.841
C01604=1163.202,414.605,-87.528,-176.136,9.575,148.841
C01605=1163.198,414.853,-87.563,-176.137,9.577,148.842
C01606=1163.194,415.100,-87.600,-176.137,9.579,148.843
C01607=1163.192,415.348,-87.637,-176.137,9.581,148.843
C01608=1163.189,415.595,-87.674,-176.138,9.582,148.844
C01609=1163.187,415.842,-87.710,-176.138,9.584,148.844
C01610=1163.187,416.182,-87.759,-176.138,9.586,148.845
C01611=1163.187,416.522,-87.809,-176.139,9.588,148.846
C01612=1163.190,416.861,-87.858,-176.140,9.591,148.846
C01613=1163.193,417.199,-87.907,-176.140,9.593,148.847
C01614=1162.773,417.202,-87.953,-176.143,9.604,148.851
C01615=1162.769,416.826,-87.899,-176.142,9.602,148.850
C01616=1162.766,416.494,-87.851,-176.142,9.599,148.849
C01617=1162.765,416.162,-87.802,-176.142,9.597,148.849
C01618=1162.766,415.831,-87.754,-176.141,9.595,148.848
C01619=1162.768,415.584,-87.718,-176.141,9.593,148.847
C01620=1162.771,415.337,-87.681,-176.140,9.592,148.847
C01621=1162.773,415.089,-87.644,-176.140,9.590,148.846
C01622=1162.778,414.841,-87.608,-176.139,9.588,148.846
C01623=1162.781,414.594,-87.572,-176.139,9.586,148.845
C01624=1162.785,414.347,-87.535,-176.139,9.584,148.844
C01625=1162.789,414.100,-87.498,-176.138,9.583,148.844
C01626=1162.793,413.852,-87.463,-176.138,9.581,148.843
C01627=1162.797,413.605,-87.426,-176.137,9.579,148.843
C01628=1162.801,413.358,-87.389,-176.137,9.577,148.842
C01629=1162.804,413.111,-87.353,-176.137,9.575,148.841
C01630=1162.809,412.863,-87.317,-176.136,9.573,148.841
C01631=1162.813,412.616,-87.280,-176.136,9.572,148.840
C01632=1162.816,412.369,-87.243,-176.135,9.570,148.840
C01633=1162.820,412.121,-87.206,-176.134,9.568,148.839
C01634=1162.824,411.873,-87.170,-176.134,9.566,148.838
C01635=1162.828,411.627,-87.134,-176.134,9.564,148.838
C01636=1162.832,411.379,-87.097,-176.133,9.563,148.837
C01637=1162.836,411.132,-87.060,-176.132,9.561,148.837
C01638=1162.839,410.885,-87.025,-176.132,9.559,148.836
C01639=1162.844,410.638,-86.988,-176.131,9.558,148.836
C01640=1162.848,410.390,-86.951,-176.131,9.555,148.835
C01641=1162.851,410.143,-86.915,-176.131,9.553,148.834
C01642=1162.855,409.896,-86.878,-176.130,9.552,148.834
C01643=1162.859,409.648,-86.842,-176.130,9.550,148.833
C01644=1162.863,409.402,-86.805,-176.129,9.548,148.832
C01645=1162.867,409.154,-86.769,-176.128,9.547,148.832
C01646=1162.871,408.907,-86.733,-176.128,9.544,148.831
C01647=1162.875,408.660,-86.696,-176.127,9.542,148.830
C01648=1162.878,408.411,-86.660,-176.127,9.541,148.830
C01649=1162.882,408.164,-86.623,-176.126,9.539,148.829
C01650=1162.886,407.917,-86.586,-176.126,9.537,148.829
C01651=1162.890,407.670,-86.550,-176.125,9.536,148.828
C01652=1162.894,407.422,-86.514,-176.125,9.533,148.827
C01653=1162.898,407.175,-86.477,-176.124,9.531,148.827
C01654=1162.901,406.928,-86.441,-176.123,9.530,148.826
C01655=1162.906,406.681,-86.405,-176.123,9.528,148.825
C01656=1162.910,406.433,-86.368,-176.123,9.525,148.825
C01657=1162.913,406.187,-86.332,-176.122,9.524,148.824
C01658=1162.917,405.939,-86.295,-176.121,9.522,148.823
C01659=1162.921,405.691,-86.259,-176.121,9.520,148.823
C01660=1162.925,405.445,-86.222,-176.120,9.518,148.822
C01661=1162.929,405.197,-86.186,-176.120,9.516,148.821
C01662=1162.933,404.950,-86.150,-176.119,9.514,148.821
C01663=1162.937,404.703,-86.113,-176.118,9.512,148.820
C01664=1162.941,404.456,-86.076,-176.118,9.511,148.819
C01665=1162.944,404.207,-86.040,-176.117,9.508,148.819
C01666=1162.948,403.960,-86.003,-176.117,9.506,148.818
C01667=1162.951,403.713,-85.967,-176.116,9.505,148.817
C01668=1162.956,403.465,-85.931,-176.116,9.502,148.817
C01669=1162.960,403.218,-85.894,-176.115,9.500,148.816
C01670=1162.963,402.971,-85.858,-176.114,9.498,148.815
C01671=1162.968,402.724,-85.822,-176.114,9.496,148.815
C01672=1162.972,402.476,-85.785,-176.113,9.494,148.814
C01673=1162.975,402.230,-85.749,-176.113,9.492,148.813
C01674=1162.979,401.982,-85.713,-176.112,9.490,148.813
C01675=1162.983,401.735,-85.676,-176.111,9.487,148.812
C01676=1162.987,401.488,-85.639,-176.111,9.486,148.811
C01677=1162.991,401.240,-85.603,-176.110,9.483,148.810
C01678=1162.995,400.993,-85.567,-176.110,9.481,148.810
C01679=1162.999,400.746,-85.530,-176.110,9.479,148.809
C01680=1163.002,400.498,-85.495,-176.108,9.477,148.808
C01681=1163.006,400.251,-85.458,-176.108,9.475,148.807
C01682=1163.011,400.004,-85.421,-176.108,9.472,148.807
C01683=1163.014,399.756,-85.385,-176.107,9.471,148.806
C01684=1163.018,399.509,-85.349,-176.106,9.468,148.805
C01685=1163.022,399.262,-85.312,-176.106,9.466,148.805
C01686=1163.026,399.014,-85.276,-176.106,9.464,148.804
C01687=1163.029,398.768,-85.240,-176.105,9.462,148.803
C01688=1163.033,398.520,-85.203,-176.104,9.459,148.802
C01689=1163.037,398.272,-85.166,-176.104,9.457,148.802
C01690=1163.041,398.025,-85.130,-176.103,9.455,148.801
C01691=1163.045,397.778,-85.093,-176.103,9.452,148.800
C01692=1163.048,397.530,-85.058,-176.102,9.450,148.799
C01693=1163.053,397.283,-85.021,-176.102,9.447,148.799
C01694=1163.057,397.035,-84.985,-176.101,9.445,148.798
C01695=1163.060,396.788,-84.949,-176.101,9.443,148.797
C01696=1163.064,396.541,-84.912,-176.101,9.440,148.796
C01697=1163.068,396.294,-84.876,-176.100,9.438,148.796
C01698=1163.072,396.047,-84.839,-176.099,9.436,148.795
C01699=1163.076,395.799,-84.804,-176.099,9.433,148.794
C01700=1163.080,395.552,-84.767,-176.099,9.430,148.793
C01701=1163.084,395.305,-84.730,-176.098,9.428,148.793
C01702=1163.088,395.057,-84.694,-176.097,9.426,148.792
C01703=1163.092,394.810,-84.658,-176.097,9.423,148.791
C01704=1163.095,394.562,-84.622,-176.097,9.420,148.790
C01705=1163.099,394.315,-84.585,-176.097,9.418,148.789
C01706=1163.103,394.068,-84.549,-176.096,9.415,148.789
C01707=1163.107,393.821,-84.513,-176.095,9.413,148.788
C01708=1163.111,393.574,-84.477,-176.095,9.410,148.787
C01709=1163.115,393.326,-84.440,-176.095,9.408,148.786
C01710=1163.118,393.079,-84.404,-176.094,9.405,148.785
C01711=1163.123,392.831,-84.368,-176.094,9.402,148.785
C01712=1163.127,392.584,-84.331,-176.094,9.400,148.784
C01713=1163.130,392.337,-84.295,-176.094,9.397,148.783
C01714=1163.135,392.089,-84.259,-176.093,9.394,148.782
C01715=1163.139,391.804,-84.217,-176.094,9.391,148.781
C01716=1163.143,391.518,-84.175,-176.093,9.388,148.781
C01717=1163.148,391.232,-84.133,-176.093,9.384,148.780
C01718=1163.152,390.948,-84.091,-176.092,9.381,148.779
C01719=1163.156,390.701,-84.056,-176.093,9.378,148.778
C01720=1163.160,390.453,-84.019,-176.093,9.375,148.777
C01721=1163.164,390.206,-83.984,-176.092,9.372,148.776
C01722=1163.168,389.959,-83.947,-176.092,9.370,148.776
C01723=1163.172,389.711,-83.911,-176.092,9.366,148.775
C01724=1163.176,389.464,-83.874,-176.092,9.364,148.774
C01725=1163.179,389.216,-83.839,-176.092,9.360,148.773
C01726=1163.183,388.969,-83.802,-176.092,9.358,148.772
C01727=1163.187,388.722,-83.766,-176.092,9.355,148.772
C01728=1163.191,388.475,-83.729,-176.092,9.351,148.771
C01729=1163.195,388.227,-83.694,-176.092,9.349,148.770
C01730=1163.199,387.980,-83.657,-176.092,9.345,148.769
C01731=1163.203,387.732,-83.621,-176.093,9.342,148.768
C01732=1163.207,387.485,-83.585,-176.092,9.339,148.768
C01733=1163.210,387.238,-83.549,-176.093,9.336,148.767
C01734=1163.214,386.991,-83.512,-176.093,9.332,148.766
C01735=1163.218,386.743,-83.477,-176.093,9.330,148.765
C01736=1163.221,386.496,-83.440,-176.093,9.326,148.765
C01737=1163.226,386.248,-83.404,-176.094,9.323,148.764
C01738=1163.230,386.001,-83.369,-176.094,9.320,148.763
C01739=1163.234,385.754,-83.332,-176.095,9.316,148.762
C01740=1163.237,385.506,-83.296,-176.095,9.313,148.761
C01741=1163.241,385.259,-83.259,-176.096,9.309,148.761
C01742=1163.245,385.011,-83.224,-176.096,9.306,148.760
C01743=1163.249,384.764,-83.188,-176.096,9.303,148.759
C01744=1163.253,384.517,-83.152,-176.097,9.299,148.758
C01745=1163.256,384.269,-83.116,-176.097,9.296,148.758
C01746=1163.261,384.021,-83.080,-176.098,9.292,148.757
C01747=1163.264,383.775,-83.044,-176.098,9.289,148.756
C01748=1163.269,383.527,-83.008,-176.099,9.286,148.756
C01749=1163.273,383.280,-82.972,-176.100,9.282,148.755
C01750=1163.276,383.033,-82.936,-176.100,9.278,148.754
C01751=1163.281,382.785,-82.900,-176.101,9.275,148.753
C01752=1163.284,382.538,-82.864,-176.102,9.272,148.753
C01753=1163.288,382.291,-82.828,-176.103,9.268,148.752
C01754=1163.292,382.043,-82.792,-176.103,9.264,148.751
C01755=1163.296,381.796,-82.756,-176.104,9.261,148.750
C01756=1163.300,381.548,-82.719,-176.105,9.257,148.750
C01757=1163.303,381.301,-82.684,-176.106,9.254,148.749
C01758=1163.307,381.053,-82.648,-176.107,9.250,148.748
C01759=1163.312,380.806,-82.613,-176.108,9.247,148.748
C01760=1163.316,380.559,-82.577,-176.109,9.242,148.747
C01761=1163.319,380.312,-82.541,-176.110,9.239,148.746
C01762=1163.324,380.064,-82.505,-176.111,9.235,148.746
C01763=1163.327,379.817,-82.469,-176.112,9.231,148.745
C01764=1163.331,379.569,-82.434,-176.113,9.228,148.744
C01765=1163.335,379.322,-82.398,-176.114,9.224,148.744
C01766=1163.339,379.074,-82.361,-176.115,9.220,148.743
C01767=1163.343,378.828,-82.326,-176.116,9.217,148.742
C01768=1163.347,378.580,-82.290,-176.118,9.213,148.742
C01769=1163.351,378.332,-82.254,-176.119,9.209,148.741
C01770=1163.355,378.085,-82.219,-176.120,9.206,148.740
C01771=1163.358,377.837,-82.183,-176.121,9.202,148.740
C01772=1163.362,377.590,-82.148,-176.123,9.198,148.739
C01773=1163.366,377.343,-82.111,-176.124,9.194,148.739
C01774=1163.370,377.096,-82.076,-176.126,9.190,148.738
C01775=1163.374,376.848,-82.040,-176.127,9.187,148.737
C01776=1163.378,376.601,-82.004,-176.128,9.183,148.737
C01777=1163.382,376.353,-81.968,-176.130,9.180,148.736
C01778=1163.386,376.105,-81.933,-176.131,9.176,148.735
C01779=1163.390,375.859,-81.898,-176.132,9.172,148.735
C01780=1163.394,375.611,-81.862,-176.134,9.168,148.734
C01781=1163.397,375.364,-81.827,-176.136,9.164,148.734
C01782=1163.402,375.116,-81.790,-176.137,9.160,148.733
C01783=1163.405,374.868,-81.755,-176.139,9.156,148.733
C01784=1163.409,374.621,-81.719,-176.140,9.153,148.732
C01785=1163.413,374.374,-81.684,-176.142,9.149,148.731
C01786=1163.417,374.127,-81.649,-176.143,9.145,148.731
C01787=1163.421,373.879,-81.613,-176.145,9.141,148.730
C01788=1163.425,373.631,-81.577,-176.147,9.138,148.730
C01789=1163.430,373.384,-81.542,-176.149,9.133,148.729
C01790=1163.433,373.136,-81.507,-176.150,9.129,148.729
C01791=1163.437,372.889,-81.471,-176.152,9.126,148.728
C01792=1163.441,372.641,-81.436,-176.154,9.122,148.728
C01793=1163.444,372.394,-81.400,-176.156,9.118,148.727
C01794=1163.449,372.147,-81.365,-176.158,9.115,148.727
C01795=1163.452,371.900,-81.329,-176.160,9.110,148.726
C01796=1163.456,371.651,-81.295,-176.161,9.106,148.726
C01797=1163.461,371.404,-81.259,-176.163,9.103,148.725
C01798=1163.465,371.157,-81.223,-176.165,9.099,148.725
C01799=1163.468,370.909,-81.188,-176.167,9.095,148.724
C01800=1163.472,370.662,-81.152,-176.169,9.091,148.724
C01801=1163.477,370.414,-81.118,-176.171,9.087,148.723
C01802=1163.480,370.167,-81.082,-176.173,9.083,148.723
C01803=1163.484,369.919,-81.047,-176.175,9.080,148.722
C01804=1163.488,369.672,-81.011,-176.177,9.075,148.722
C01805=1163.492,369.424,-80.977,-176.178,9.072,148.721
C01806=1163.496,369.177,-80.941,-176.180,9.068,148.721
C01807=1163.500,368.929,-80.906,-176.183,9.064,148.720
C01808=1163.504,368.682,-80.871,-176.185,9.060,148.720
C01809=1163.508,368.435,-80.836,-176.187,9.056,148.720
C01810=1163.511,368.187,-80.800,-176.189,9.052,148.719
C01811=1163.516,367.940,-80.766,-176.191,9.049,148.719
C01812=1163.520,367.692,-80.730,-176.193,9.045,148.718
C01813=1163.524,367.444,-80.695,-176.196,9.041,148.718
C01814=1163.528,367.197,-80.660,-176.197,9.037,148.718
C01815=1163.531,366.950,-80.625,-176.200,9.033,148.717
